KUKA KRL program: EPS_2_251806_MH48A_A_20260212042246.src

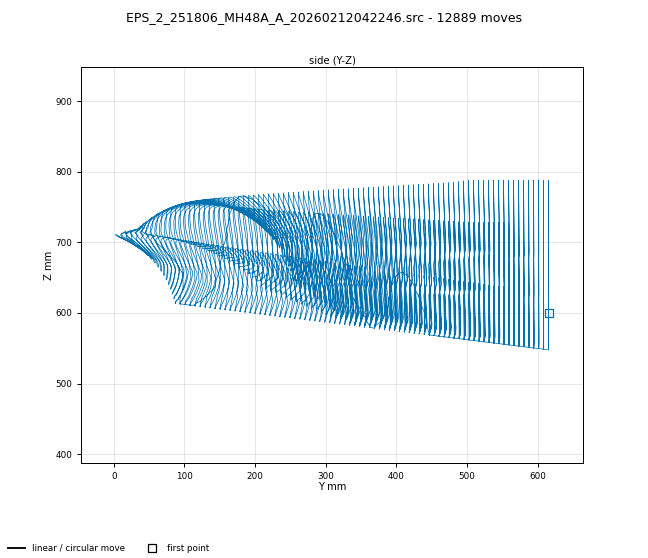
[picture p0: tool path of EPS_2_251806_MH48A_A_20260212042246.src, 12889 of 12891 moves have a stored position in this frame; points joined in program order, loops and branches not executed]
&ACCESS RVP
&REL 4
&COMMENT QRS 19112012
&PARAM EDITMASK = *
DEF PART()
EXT BAS (BAS_COMMAND :IN,REAL :IN )
INT I
BAS (#INITMOV,0 )

;KUKA QRS Post kuka4.cps  Date:22-06-2017 !

File_ID=3020

QRS_PRE_INIT()

;Init var - Until changes are made in qrs_pre_init
Outlet_Square_prg=0
Inlet_1_Square_prg=0
Inlet_2_Square_prg=0
Inlet_3_Square_prg=0
Inlet_4_Square_prg=0
Inlet_5_Square_prg=0

Outlet_1={X 0.000, Y 504.220, Z 687.500, B 0.000, E1 0.000 }
Inlet_1={X 0.000, Y 539.050, Z 207.500, B 0.000, E1 194.000 }
Inlet_2={X 0.000, Y 508.580, Z 627.500, B 0.000, E1 257.000 }
Outlet_1_type=201
Inlet_1_type=201
Inlet_2_type=201
;QRS#1=Sidecore dimensions
;QRS#2=200-8" PVC SDR 35
;QRS#3=200-8" PVC SDR 35
;QRS#4=200-8" PVC SDR 35
;QRS#5=
;QRS#6=
;QRS#7=
;QRS#8=
;QRS#9=12-08 PSX
;QRS#10=12-08 PSX
;QRS#11=12-08 PSX
;QRS#12=
;QRS#13=
;QRS#14=
;QRS#15=
;QRS#16=1220x127x1067 3,5'
;QRS#17=EPS Height
;QRS#18=788
;QRS#19=*
;QRS#20= UPDATED VERSION 22-06-2017
;QRS#21=*
Outlet_Square=0100
Inlet_1_Square=0100
Inlet_2_Square=0100
Inlet_3_Square=0
Inlet_4_Square=0
Inlet_5_Square=0
Mill_Square=1
Outlet_Square_Prg=204
Inlet_1_Square_prg=204
Inlet_2_Square_prg=204

QRS_INIT()

$ADVANCE=5

; T1
PTP {E1 173.607,E2 173.607}
PTP {X 0,Y 615.504,A -85,B 0,C 180,E1 173.607,E2 173.607,E3 0,E4 0,E5 0,E6 0}
QRS_SPEED_INIT()
LIN {X 0,Y 615.504,Z 600,A -85,B 0,C 180,E1 173.607,E2 173.607,E3 0,E4 0,E5 0,E6 0} C_VEL
LIN {X 0,Y 615.504,Z 557.872,A -85,B 0,C 180,E1 173.607,E2 173.607} C_VEL
LIN {X 0,Y 615.504,Z 549.695,A -85,B 0,C 180,E1 173.607,E2 173.607} C_VEL
LIN {X 0,Y 615.491,Z 547.695,A -85,B 0,C 180,E1 173.421,E2 173.421} C_VEL
LIN {X 0,Y 615.488,Z 547.7,A -85,B 0,C 180,E1 170.801,E2 170.801} C_VEL
LIN {X 0,Y 615.487,Z 547.699,A -85,B 0,C 180,E1 168.139,E2 168.139} C_VEL
LIN {X 0,Y 615.487,Z 547.696,A -85,B 0,C 180,E1 165.451,E2 165.451} C_VEL
LIN {X 0,Y 615.478,Z 547.7,A -85,B 0,C 180,E1 162.73,E2 162.73} C_VEL
LIN {X 0,Y 615.483,Z 547.7,A -85,B 0,C 180,E1 159.967,E2 159.967} C_VEL
LIN {X 0,Y 615.482,Z 547.697,A -85,B 0,C 180,E1 157.156,E2 157.156} C_VEL
LIN {X 0,Y 615.498,Z 547.7,A -85,B 0,C 180,E1 154.285,E2 154.285} C_VEL
LIN {X 0,Y 615.485,Z 547.696,A -85,B 0,C 180,E1 151.342,E2 151.342} C_VEL
LIN {X 0,Y 615.477,Z 547.698,A -85,B 0,C 180,E1 148.916,E2 148.916} C_VEL
LIN {X 0,Y 615.486,Z 547.697,A -85,B 0,C 180,E1 146.466,E2 146.466} C_VEL
LIN {X 0,Y 615.491,Z 547.698,A -85,B 0,C 180,E1 143.576,E2 143.576} C_VEL
LIN {X 0,Y 615.479,Z 547.698,A -85,B 0,C 180,E1 140.939,E2 140.939} C_VEL
LIN {X 0,Y 615.486,Z 547.696,A -85,B 0,C 180,E1 138.526,E2 138.526} C_VEL
LIN {X 0,Y 615.489,Z 547.698,A -85,B 0,C 180,E1 135.851,E2 135.851} C_VEL
LIN {X 0,Y 615.486,Z 547.699,A -85,B 0,C 180,E1 133.048,E2 133.048} C_VEL
LIN {X 0,Y 615.496,Z 547.695,A -85,B 0,C 180,E1 130.09,E2 130.09} C_VEL
LIN {X 0,Y 615.495,Z 547.697,A -85,B 0,C 180,E1 127.242,E2 127.242} C_VEL
LIN {X 0,Y 615.479,Z 547.698,A -85,B 0,C 180,E1 124.7,E2 124.7} C_VEL
LIN {X 0,Y 615.494,Z 547.695,A -85,B 0,C 180,E1 122.332,E2 122.332} C_VEL
LIN {X 0,Y 615.486,Z 547.7,A -85,B 0,C 180,E1 119.407,E2 119.407} C_VEL
LIN {X 0,Y 615.491,Z 547.699,A -85,B 0,C 180,E1 117.046,E2 117.046} C_VEL
LIN {X 0,Y 615.495,Z 547.695,A -85,B 0,C 180,E1 114.272,E2 114.272} C_VEL
LIN {X 0,Y 615.48,Z 547.699,A -85,B 0,C 180,E1 111.433,E2 111.433} C_VEL
LIN {X 0,Y 615.489,Z 547.699,A -85,B 0,C 180,E1 108.606,E2 108.606} C_VEL
LIN {X 0,Y 615.489,Z 547.695,A -85,B 0,C 180,E1 105.906,E2 105.906} C_VEL
LIN {X 0,Y 615.488,Z 547.697,A -85,B 0,C 180,E1 103.202,E2 103.202} C_VEL
LIN {X 0,Y 615.491,Z 547.701,A -85,B 0,C 180,E1 100.527,E2 100.527} C_VEL
LIN {X 0,Y 615.487,Z 547.697,A -85,B 0,C 180,E1 97.876,E2 97.876} C_VEL
LIN {X 0,Y 615.481,Z 547.697,A -85,B 0,C 180,E1 95.242,E2 95.242} C_VEL
LIN {X 0,Y 615.483,Z 547.699,A -85,B 0,C 180,E1 92.618,E2 92.618} C_VEL
LIN {X 0,Y 615.487,Z 547.702,A -85,B 0,C 180,E1 90.001,E2 90.001} C_VEL
LIN {X 0,Y 615.482,Z 547.697,A -85,B 0,C 180,E1 87.239,E2 87.239} C_VEL
LIN {X 0,Y 615.486,Z 560.488,A -85,B 0,C 180,E1 86.81,E2 86.81} C_VEL
LIN {X 0,Y 615.491,Z 571.428,A -85,B 0,C 180,E1 86.318,E2 86.318} C_VEL
LIN {X 0,Y 615.49,Z 582.825,A -85,B 0,C 180,E1 85.662,E2 85.662} C_VEL
LIN {X 0,Y 615.498,Z 593.104,A -85,B 0,C 180,E1 84.924,E2 84.924} C_VEL
LIN {X 0,Y 615.5,Z 602.425,A -85,B 0,C 180,E1 84.102,E2 84.102} C_VEL
LIN {X 0,Y 615.496,Z 611.553,A -85,B 0,C 180,E1 83.099,E2 83.099} C_VEL
LIN {X 0,Y 615.497,Z 618.702,A -85,B 0,C 180,E1 82.125,E2 82.125} C_VEL
LIN {X 0,Y 615.496,Z 624.55,A -85,B 0,C 180,E1 81.133,E2 81.133} C_VEL
LIN {X 0,Y 615.497,Z 629.163,A -85,B 0,C 180,E1 80.139,E2 80.139} C_VEL
LIN {X 0,Y 615.495,Z 632.786,A -85,B 0,C 180,E1 79.107,E2 79.107} C_VEL
LIN {X 0,Y 615.496,Z 635.183,A -85,B 0,C 180,E1 78.14,E2 78.14} C_VEL
LIN {X 0,Y 615.495,Z 636.336,A -85,B 0,C 180,E1 77.471,E2 77.471} C_VEL
LIN {X 0,Y 615.495,Z 637.353,A -85,B 0,C 180,E1 76.127,E2 76.127} C_VEL
LIN {X 0,Y 615.497,Z 637.272,A -85,B 0,C 180,E1 75.452,E2 75.452} C_VEL
LIN {X 0,Y 615.496,Z 636.732,A -85,B 0,C 180,E1 74.775,E2 74.775} C_VEL
LIN {X 0,Y 615.493,Z 634.742,A -85,B 0,C 180,E1 73.566,E2 73.566} C_VEL
LIN {X 0,Y 615.496,Z 631.457,A -85,B 0,C 180,E1 72.388,E2 72.388} C_VEL
LIN {X 0,Y 615.497,Z 627.375,A -85,B 0,C 180,E1 71.355,E2 71.355} C_VEL
LIN {X 0,Y 615.497,Z 620.947,A -85,B 0,C 180,E1 70.142,E2 70.142} C_VEL
LIN {X 0,Y 615.497,Z 613.808,A -85,B 0,C 180,E1 69.095,E2 69.095} C_VEL
LIN {X 0,Y 615.499,Z 606.411,A -85,B 0,C 180,E1 68.218,E2 68.218} C_VEL
LIN {X 0,Y 615.5,Z 598.09,A -85,B 0,C 180,E1 67.404,E2 67.404} C_VEL
LIN {X 0,Y 615.5,Z 588.32,A -85,B 0,C 180,E1 66.623,E2 66.623} C_VEL
LIN {X 0,Y 615.496,Z 577.54,A -85,B 0,C 180,E1 65.925,E2 65.925} C_VEL
LIN {X 0,Y 615.491,Z 565.819,A -85,B 0,C 180,E1 65.325,E2 65.325} C_VEL
LIN {X 0,Y 615.487,Z 553.967,A -85,B 0,C 180,E1 64.865,E2 64.865} C_VEL
LIN {X 0,Y 615.479,Z 547.698,A -85,B 0,C 180,E1 64.667,E2 64.667} C_VEL
LIN {X 0,Y 615.484,Z 547.699,A -85,B 0,C 180,E1 62.086,E2 62.086} C_VEL
LIN {X 0,Y 615.499,Z 547.695,A -85,B 0,C 180,E1 59.842,E2 59.842} C_VEL
LIN {X 0,Y 615.491,Z 547.696,A -85,B 0,C 180,E1 57.544,E2 57.544} C_VEL
LIN {X 0,Y 615.478,Z 547.699,A -85,B 0,C 180,E1 55.185,E2 55.185} C_VEL
LIN {X 0,Y 615.494,Z 547.697,A -85,B 0,C 180,E1 52.759,E2 52.759} C_VEL
LIN {X 0,Y 615.494,Z 547.696,A -85,B 0,C 180,E1 49.91,E2 49.91} C_VEL
LIN {X 0,Y 615.482,Z 547.787,A -85,B 0,C 180,E1 48.147,E2 48.147} C_VEL
LIN {X 0,Y 615.494,Z 554.573,A -85,B 0,C 180,E1 45.852,E2 45.852} C_VEL
LIN {X 0,Y 615.482,Z 562.723,A -85,B 0,C 180,E1 43.048,E2 43.048} C_VEL
LIN {X 0,Y 615.484,Z 570.001,A -85,B 0,C 180,E1 40.606,E2 40.606} C_VEL
LIN {X 0,Y 615.48,Z 577.917,A -85,B 0,C 180,E1 38.013,E2 38.013} C_VEL
LIN {X 0,Y 615.478,Z 586.629,A -85,B 0,C 180,E1 35.215,E2 35.215} C_VEL
LIN {X 0,Y 615.484,Z 595.394,A -85,B 0,C 180,E1 32.457,E2 32.457} C_VEL
LIN {X 0,Y 615.498,Z 603.966,A -85,B 0,C 180,E1 29.798,E2 29.798} C_VEL
LIN {X 0,Y 615.478,Z 612.988,A -85,B 0,C 180,E1 27.045,E2 27.045} C_VEL
LIN {X 0,Y 615.492,Z 621.119,A -85,B 0,C 180,E1 24.586,E2 24.586} C_VEL
LIN {X 0,Y 615.492,Z 634.761,A -85,B 0,C 180,E1 24.316,E2 24.316} C_VEL
LIN {X 0,Y 615.486,Z 646.624,A -85,B 0,C 180,E1 23.953,E2 23.953} C_VEL
LIN {X 0,Y 615.484,Z 658.337,A -85,B 0,C 180,E1 23.467,E2 23.467} C_VEL
LIN {X 0,Y 615.481,Z 669.928,A -85,B 0,C 180,E1 22.844,E2 22.844} C_VEL
LIN {X 0,Y 615.499,Z 680.403,A -85,B 0,C 180,E1 22.136,E2 22.136} C_VEL
LIN {X 0,Y 615.497,Z 690.798,A -85,B 0,C 180,E1 21.256,E2 21.256} C_VEL
LIN {X 0,Y 615.496,Z 699.931,A -85,B 0,C 180,E1 20.297,E2 20.297} C_VEL
LIN {X 0,Y 615.498,Z 707.268,A -85,B 0,C 180,E1 19.337,E2 19.337} C_VEL
LIN {X 0,Y 615.498,Z 713.727,A -85,B 0,C 180,E1 18.283,E2 18.283} C_VEL
LIN {X 0,Y 615.495,Z 718.599,A -85,B 0,C 180,E1 17.27,E2 17.27} C_VEL
LIN {X 0,Y 615.495,Z 721.729,A -85,B 0,C 180,E1 16.437,E2 16.437} C_VEL
LIN {X 0,Y 615.496,Z 724.998,A -85,B 0,C 180,E1 15.226,E2 15.226} C_VEL
LIN {X 0,Y 615.494,Z 726.224,A -85,B 0,C 180,E1 14.549,E2 14.549} C_VEL
LIN {X 0,Y 615.494,Z 726.988,A -85,B 0,C 180,E1 13.874,E2 13.874} C_VEL
LIN {X 0,Y 615.494,Z 727.294,A -85,B 0,C 180,E1 12.53,E2 12.53} C_VEL
LIN {X 0,Y 615.495,Z 726.833,A -85,B 0,C 180,E1 11.86,E2 11.86} C_VEL
LIN {X 0,Y 615.493,Z 725.447,A -85,B 0,C 180,E1 10.896,E2 10.896} C_VEL
LIN {X 0,Y 615.499,Z 721.91,A -85,B 0,C 180,E1 9.53,E2 9.53} C_VEL
LIN {X 0,Y 615.495,Z 718.153,A -85,B 0,C 180,E1 8.536,E2 8.536} C_VEL
LIN {X 0,Y 615.498,Z 713.28,A -85,B 0,C 180,E1 7.545,E2 7.545} C_VEL
LIN {X 0,Y 615.496,Z 707.157,A -85,B 0,C 180,E1 6.556,E2 6.556} C_VEL
LIN {X 0,Y 615.499,Z 699.561,A -85,B 0,C 180,E1 5.569,E2 5.569} C_VEL
LIN {X 0,Y 615.497,Z 690.049,A -85,B 0,C 180,E1 4.584,E2 4.584} C_VEL
LIN {X 0,Y 615.5,Z 680.271,A -85,B 0,C 180,E1 3.764,E2 3.764} C_VEL
LIN {X 0,Y 615.479,Z 669.277,A -85,B 0,C 180,E1 3.027,E2 3.027} C_VEL
LIN {X 0,Y 615.489,Z 658.562,A -85,B 0,C 180,E1 2.454,E2 2.454} C_VEL
LIN {X 0,Y 615.477,Z 646.799,A -85,B 0,C 180,E1 1.963,E2 1.963} C_VEL
LIN {X 0,Y 615.487,Z 634.805,A -85,B 0,C 180,E1 1.595,E2 1.595} C_VEL
LIN {X 0,Y 615.488,Z 622.794,A -85,B 0,C 180,E1 1.349,E2 1.349} C_VEL
LIN {X 0,Y 615.485,Z 621.087,A -85,B 0,C 180,E1 1.308,E2 1.308} C_VEL
LIN {X 0,Y 615.485,Z 612.466,A -85,B 0,C 180,E1 -1.309,E2 -1.309} C_VEL
LIN {X 0,Y 615.49,Z 603.925,A -85,B 0,C 180,E1 -3.929,E2 -3.929} C_VEL
LIN {X 0,Y 615.489,Z 595.382,A -85,B 0,C 180,E1 -6.589,E2 -6.589} C_VEL
LIN {X 0,Y 615.496,Z 586.076,A -85,B 0,C 180,E1 -9.53,E2 -9.53} C_VEL
LIN {X 0,Y 615.475,Z 577.824,A -85,B 0,C 180,E1 -12.196,E2 -12.196} C_VEL
LIN {X 0,Y 615.492,Z 569.65,A -85,B 0,C 180,E1 -14.887,E2 -14.887} C_VEL
LIN {X 0,Y 615.499,Z 561.583,A -85,B 0,C 180,E1 -17.613,E2 -17.613} C_VEL
LIN {X 0,Y 615.489,Z 553.106,A -85,B 0,C 180,E1 -20.56,E2 -20.56} C_VEL
LIN {X 0,Y 615.497,Z 549.253,A -85,B 0,C 180,E1 -21.784,E2 -21.784} C_VEL
LIN {X 0,Y 615.484,Z 547.698,A -85,B 0,C 180,E1 -22.243,E2 -22.243} C_VEL
LIN {X 0,Y 615.492,Z 547.701,A -85,B 0,C 180,E1 -24.992,E2 -24.992} C_VEL
LIN {X 0,Y 615.492,Z 547.699,A -85,B 0,C 180,E1 -27.915,E2 -27.915} C_VEL
LIN {X 0,Y 615.5,Z 547.7,A -85,B 0,C 180,E1 -30.16,E2 -30.16} C_VEL
LIN {X 0,Y 615.495,Z 547.697,A -85,B 0,C 180,E1 -32.457,E2 -32.457} C_VEL
LIN {X 0,Y 615.494,Z 547.696,A -85,B 0,C 180,E1 -34.815,E2 -34.815} C_VEL
LIN {X 0,Y 615.49,Z 547.699,A -85,B 0,C 180,E1 -37.242,E2 -37.242} C_VEL
LIN {X 0,Y 615.479,Z 547.699,A -85,B 0,C 180,E1 -40.09,E2 -40.09} C_VEL
LIN {X 0,Y 615.485,Z 547.699,A -85,B 0,C 180,E1 -42.354,E2 -42.354} C_VEL
LIN {X 0,Y 615.481,Z 547.699,A -85,B 0,C 180,E1 -45.069,E2 -45.069} C_VEL
LIN {X 0,Y 615.488,Z 547.7,A -85,B 0,C 180,E1 -47.92,E2 -47.92} C_VEL
LIN {X 0,Y 615.48,Z 547.699,A -85,B 0,C 180,E1 -50.25,E2 -50.25} C_VEL
LIN {X 0,Y 615.49,Z 547.7,A -85,B 0,C 180,E1 -53.063,E2 -53.063} C_VEL
LIN {X 0,Y 615.484,Z 547.718,A -85,B 0,C 180,E1 -54.486,E2 -54.486} C_VEL
LIN {X 0,Y 615.49,Z 561.14,A -85,B 0,C 180,E1 -57.155,E2 -57.155} C_VEL
LIN {X 0,Y 615.499,Z 574.889,A -85,B 0,C 180,E1 -59.842,E2 -59.842} C_VEL
LIN {X 0,Y 615.488,Z 590.604,A -85,B 0,C 180,E1 -62.824,E2 -62.824} C_VEL
LIN {X 0,Y 615.488,Z 606.309,A -85,B 0,C 180,E1 -65.729,E2 -65.729} C_VEL
LIN {X 0,Y 615.486,Z 622.001,A -85,B 0,C 180,E1 -68.569,E2 -68.569} C_VEL
LIN {X 0,Y 615.479,Z 637.926,A -85,B 0,C 180,E1 -71.399,E2 -71.399} C_VEL
LIN {X 0,Y 615.495,Z 653.333,A -85,B 0,C 180,E1 -74.096,E2 -74.096} C_VEL
LIN {X 0,Y 615.488,Z 668.981,A -85,B 0,C 180,E1 -76.8,E2 -76.8} C_VEL
LIN {X 0,Y 615.478,Z 678,A -85,B 0,C 180,E1 -78.328,E2 -78.328} C_VEL
LIN {X 0,Y 615.478,Z 691.273,A -85,B 0,C 180,E1 -78.557,E2 -78.557} C_VEL
LIN {X 0,Y 615.499,Z 704.348,A -85,B 0,C 180,E1 -78.923,E2 -78.923} C_VEL
LIN {X 0,Y 615.476,Z 716.143,A -85,B 0,C 180,E1 -79.384,E2 -79.384} C_VEL
LIN {X 0,Y 615.488,Z 727.587,A -85,B 0,C 180,E1 -79.972,E2 -79.972} C_VEL
LIN {X 0,Y 615.499,Z 739.031,A -85,B 0,C 180,E1 -80.719,E2 -80.719} C_VEL
LIN {X 0,Y 615.498,Z 748.265,A -85,B 0,C 180,E1 -81.464,E2 -81.464} C_VEL
LIN {X 0,Y 615.499,Z 756.659,A -85,B 0,C 180,E1 -82.29,E2 -82.29} C_VEL
LIN {X 0,Y 615.497,Z 764.692,A -85,B 0,C 180,E1 -83.259,E2 -83.259} C_VEL
LIN {X 0,Y 615.498,Z 770.427,A -85,B 0,C 180,E1 -84.102,E2 -84.102} C_VEL
LIN {X 0,Y 615.497,Z 775.875,A -85,B 0,C 180,E1 -85.088,E2 -85.088} C_VEL
LIN {X 0,Y 615.496,Z 780.143,A -85,B 0,C 180,E1 -86.072,E2 -86.072} C_VEL
LIN {X 0,Y 615.495,Z 782.401,A -85,B 0,C 180,E1 -86.728,E2 -86.728} C_VEL
LIN {X 0,Y 615.497,Z 784.234,A -85,B 0,C 180,E1 -87.383,E2 -87.383} C_VEL
LIN {X 0,Y 615.496,Z 785.609,A -85,B 0,C 180,E1 -88.038,E2 -88.038} C_VEL
LIN {X 0,Y 615.496,Z 787.174,A -85,B 0,C 180,E1 -89.346,E2 -89.346} C_VEL
LIN {X 0,Y 615.494,Z 787.389,A -85,B 0,C 180,E1 -90.001,E2 -90.001} C_VEL
LIN {X 0,Y 615.496,Z 786.579,A -85,B 0,C 180,E1 -91.309,E2 -91.309} C_VEL
LIN {X 0,Y 615.496,Z 785.607,A -85,B 0,C 180,E1 -91.964,E2 -91.964} C_VEL
LIN {X 0,Y 615.497,Z 784.231,A -85,B 0,C 180,E1 -92.618,E2 -92.618} C_VEL
LIN {X 0,Y 615.496,Z 781.348,A -85,B 0,C 180,E1 -93.601,E2 -93.601} C_VEL
LIN {X 0,Y 615.498,Z 777.439,A -85,B 0,C 180,E1 -94.585,E2 -94.585} C_VEL
LIN {X 0,Y 615.499,Z 772.402,A -85,B 0,C 180,E1 -95.57,E2 -95.57} C_VEL
LIN {X 0,Y 615.497,Z 765.87,A -85,B 0,C 180,E1 -96.583,E2 -96.583} C_VEL
LIN {X 0,Y 615.497,Z 758.128,A -85,B 0,C 180,E1 -97.546,E2 -97.546} C_VEL
LIN {X 0,Y 615.498,Z 750.039,A -85,B 0,C 180,E1 -98.372,E2 -98.372} C_VEL
LIN {X 0,Y 615.499,Z 740.16,A -85,B 0,C 180,E1 -99.199,E2 -99.199} C_VEL
LIN {X 0,Y 615.486,Z 728.973,A -85,B 0,C 180,E1 -99.946,E2 -99.946} C_VEL
LIN {X 0,Y 615.476,Z 718.013,A -85,B 0,C 180,E1 -100.528,E2 -100.528} C_VEL
LIN {X 0,Y 615.497,Z 705.495,A -85,B 0,C 180,E1 -101.04,E2 -101.04} C_VEL
LIN {X 0,Y 615.479,Z 693.044,A -85,B 0,C 180,E1 -101.402,E2 -101.402} C_VEL
LIN {X 0,Y 615.477,Z 679.431,A -85,B 0,C 180,E1 -101.653,E2 -101.653} C_VEL
LIN {X 0,Y 615.478,Z 677.795,A -85,B 0,C 180,E1 -101.694,E2 -101.694} C_VEL
LIN {X 0,Y 615.491,Z 663.028,A -85,B 0,C 180,E1 -104.24,E2 -104.24} C_VEL
LIN {X 0,Y 615.487,Z 647.605,A -85,B 0,C 180,E1 -106.929,E2 -106.929} C_VEL
LIN {X 0,Y 615.476,Z 632.002,A -85,B 0,C 180,E1 -109.686,E2 -109.686} C_VEL
LIN {X 0,Y 615.48,Z 617.194,A -85,B 0,C 180,E1 -112.344,E2 -112.344} C_VEL
LIN {X 0,Y 615.494,Z 602.704,A -85,B 0,C 180,E1 -114.992,E2 -114.992} C_VEL
LIN {X 0,Y 615.48,Z 589.015,A -85,B 0,C 180,E1 -117.546,E2 -117.546} C_VEL
LIN {X 0,Y 615.499,Z 575.32,A -85,B 0,C 180,E1 -120.16,E2 -120.16} C_VEL
LIN {X 0,Y 615.491,Z 561.625,A -85,B 0,C 180,E1 -122.846,E2 -122.846} C_VEL
LIN {X 0,Y 615.475,Z 547.698,A -85,B 0,C 180,E1 -125.644,E2 -125.644} C_VEL
LIN {X 0,Y 615.489,Z 547.695,A -85,B 0,C 180,E1 -128.069,E2 -128.069} C_VEL
LIN {X 0,Y 615.481,Z 547.698,A -85,B 0,C 180,E1 -130.607,E2 -130.607} C_VEL
LIN {X 0,Y 615.499,Z 547.7,A -85,B 0,C 180,E1 -133.244,E2 -133.244} C_VEL
LIN {X 0,Y 615.485,Z 547.697,A -85,B 0,C 180,E1 -136.003,E2 -136.003} C_VEL
LIN {X 0,Y 615.486,Z 547.699,A -85,B 0,C 180,E1 -138.906,E2 -138.906} C_VEL
LIN {X 0,Y 615.484,Z 547.698,A -85,B 0,C 180,E1 -141.095,E2 -141.095} C_VEL
LIN {X 0,Y 615.495,Z 547.697,A -85,B 0,C 180,E1 -143.575,E2 -143.575} C_VEL
LIN {X 0,Y 615.489,Z 547.699,A -85,B 0,C 180,E1 -145.978,E2 -145.978} C_VEL
LIN {X 0,Y 615.49,Z 547.699,A -85,B 0,C 180,E1 -148.314,E2 -148.314} C_VEL
LIN {X 0,Y 615.482,Z 547.7,A -85,B 0,C 180,E1 -150.593,E2 -150.593} C_VEL
LIN {X 0,Y 615.487,Z 547.699,A -85,B 0,C 180,E1 -152.955,E2 -152.955} C_VEL
LIN {X 0,Y 615.482,Z 547.699,A -85,B 0,C 180,E1 -155.727,E2 -155.727} C_VEL
LIN {X 0,Y 615.486,Z 547.697,A -85,B 0,C 180,E1 -158.568,E2 -158.568} C_VEL
LIN {X 0,Y 615.493,Z 547.7,A -85,B 0,C 180,E1 -161.394,E2 -161.394} C_VEL
LIN {X 0,Y 615.48,Z 547.698,A -85,B 0,C 180,E1 -164.094,E2 -164.094} C_VEL
LIN {X 0,Y 615.479,Z 547.699,A -85,B 0,C 180,E1 -166.798,E2 -166.798} C_VEL
LIN {X 0,Y 615.49,Z 547.702,A -85,B 0,C 180,E1 -169.473,E2 -169.473} C_VEL
LIN {X 0,Y 615.483,Z 547.698,A -85,B 0,C 180,E1 -172.124,E2 -172.124} C_VEL
LIN {X 0,Y 615.481,Z 547.697,A -85,B 0,C 180,E1 -174.758,E2 -174.758} C_VEL
LIN {X 0,Y 615.492,Z 547.697,A -85,B 0,C 180,E1 -177.382,E2 -177.382} C_VEL
LIN {X 0,Y 615.489,Z 547.703,A -85,B 0,C 180,E1 -180,E2 -180} C_VEL
LIN {X 0,Y 615.492,Z 547.697,A -85,B 0,C 180,E1 -182.618,E2 -182.618} C_VEL
LIN {X 0,Y 615.481,Z 547.697,A -85,B 0,C 180,E1 -185.241,E2 -185.241} C_VEL
LIN {X 0,Y 615.491,Z 547.695,A -85,B 0,C 180,E1 -186.579,E2 -186.579} C_VEL
LIN {X 0,Y 614.815,Z 547.844,A -85,B 0,C 180,E1 -187.125,E2 -187.125} C_VEL
LIN {X 0,Y 611.981,Z 548.257,A -85,B 0,C 180,E1 -188.011,E2 -188.011} C_VEL
LIN {X 0,Y 609.587,Z 548.568,A -85,B 0,C 180,E1 -188.724,E2 -188.724} C_VEL
LIN {X 0,Y 608.549,Z 548.687,A -85,B 0,C 180,E1 -189.273,E2 -189.273} C_VEL
LIN {X 0,Y 608.458,Z 548.696,A -85,B 0,C 180,E1 -189.46,E2 -189.46} C_VEL
LIN {X 0,Y 608.464,Z 548.694,A -85,B 0,C 180,E1 -191.999,E2 -191.999} C_VEL
LIN {X 0,Y 608.478,Z 548.692,A -85,B 0,C 180,E1 -194.72,E2 -194.72} C_VEL
LIN {X 0,Y 608.446,Z 548.699,A -85,B 0,C 180,E1 -197.476,E2 -197.476} C_VEL
LIN {X 0,Y 608.45,Z 548.696,A -85,B 0,C 180,E1 -199.57,E2 -199.57} C_VEL
LIN {X 0,Y 608.46,Z 548.695,A -85,B 0,C 180,E1 -202.476,E2 -202.476} C_VEL
LIN {X 0,Y 608.45,Z 548.698,A -85,B 0,C 180,E1 -204.571,E2 -204.571} C_VEL
LIN {X 0,Y 608.481,Z 548.692,A -85,B 0,C 180,E1 -207.207,E2 -207.207} C_VEL
LIN {X 0,Y 608.471,Z 548.693,A -85,B 0,C 180,E1 -209.972,E2 -209.972} C_VEL
LIN {X 0,Y 608.453,Z 548.696,A -85,B 0,C 180,E1 -212.879,E2 -212.879} C_VEL
LIN {X 0,Y 608.449,Z 548.696,A -85,B 0,C 180,E1 -215.277,E2 -215.277} C_VEL
LIN {X 0,Y 608.469,Z 548.693,A -85,B 0,C 180,E1 -217.746,E2 -217.746} C_VEL
LIN {X 0,Y 608.446,Z 548.695,A -85,B 0,C 180,E1 -220.328,E2 -220.328} C_VEL
LIN {X 0,Y 608.453,Z 548.696,A -85,B 0,C 180,E1 -222.959,E2 -222.959} C_VEL
LIN {X 0,Y 608.46,Z 548.695,A -85,B 0,C 180,E1 -225.735,E2 -225.735} C_VEL
LIN {X 0,Y 608.464,Z 548.694,A -85,B 0,C 180,E1 -228.657,E2 -228.657} C_VEL
LIN {X 0,Y 608.469,Z 548.696,A -85,B 0,C 180,E1 -231.412,E2 -231.412} C_VEL
LIN {X 0,Y 608.445,Z 548.697,A -85,B 0,C 180,E1 -233.954,E2 -233.954} C_VEL
LIN {X 0,Y 608.463,Z 548.694,A -85,B 0,C 180,E1 -236.329,E2 -236.329} C_VEL
LIN {X 0,Y 608.479,Z 548.692,A -85,B 0,C 180,E1 -238.727,E2 -238.727} C_VEL
LIN {X 0,Y 608.467,Z 548.693,A -85,B 0,C 180,E1 -241.381,E2 -241.381} C_VEL
LIN {X 0,Y 608.451,Z 548.696,A -85,B 0,C 180,E1 -243.964,E2 -243.964} C_VEL
LIN {X 0,Y 608.472,Z 548.692,A -85,B 0,C 180,E1 -246.155,E2 -246.155} C_VEL
LIN {X 0,Y 608.468,Z 548.693,A -85,B 0,C 180,E1 -248.308,E2 -248.308} C_VEL
LIN {X 0,Y 608.473,Z 548.696,A -85,B 0,C 180,E1 -251.283,E2 -251.283} C_VEL
LIN {X 0,Y 608.464,Z 548.694,A -85,B 0,C 180,E1 -253.906,E2 -253.906} C_VEL
LIN {X 0,Y 608.465,Z 548.693,A -85,B 0,C 180,E1 -256.643,E2 -256.643} C_VEL
LIN {X 0,Y 608.468,Z 548.695,A -85,B 0,C 180,E1 -259.35,E2 -259.35} C_VEL
LIN {X 0,Y 608.478,Z 548.693,A -85,B 0,C 180,E1 -262.033,E2 -262.033} C_VEL
LIN {X 0,Y 608.462,Z 548.693,A -85,B 0,C 180,E1 -264.698,E2 -264.698} C_VEL
LIN {X 0,Y 608.475,Z 548.693,A -85,B 0,C 180,E1 -267.351,E2 -267.351} C_VEL
LIN {X 0,Y 608.478,Z 548.695,A -85,B 0,C 180,E1 -269.999,E2 -269.999} C_VEL
LIN {X 0,Y 608.472,Z 548.693,A -85,B 0,C 180,E1 -272.647,E2 -272.647} C_VEL
LIN {X 0,Y 608.506,Z 562.528,A -85,B 0,C 180,E1 -273.144,E2 -273.144} C_VEL
LIN {X 0,Y 608.512,Z 574.619,A -85,B 0,C 180,E1 -273.724,E2 -273.724} C_VEL
LIN {X 0,Y 608.479,Z 585.509,A -85,B 0,C 180,E1 -274.388,E2 -274.388} C_VEL
LIN {X 0,Y 608.482,Z 595.356,A -85,B 0,C 180,E1 -275.135,E2 -275.135} C_VEL
LIN {X 0,Y 608.456,Z 604.326,A -85,B 0,C 180,E1 -275.966,E2 -275.966} C_VEL
LIN {X 0,Y 608.462,Z 613.118,A -85,B 0,C 180,E1 -276.965,E2 -276.965} C_VEL
LIN {X 0,Y 608.44,Z 620.192,A -85,B 0,C 180,E1 -277.967,E2 -277.967} C_VEL
LIN {X 0,Y 608.446,Z 625.856,A -85,B 0,C 180,E1 -278.97,E2 -278.97} C_VEL
LIN {X 0,Y 608.436,Z 630.327,A -85,B 0,C 180,E1 -279.977,E2 -279.977} C_VEL
LIN {X 0,Y 608.452,Z 633.614,A -85,B 0,C 180,E1 -280.949,E2 -280.949} C_VEL
LIN {X 0,Y 608.439,Z 636.102,A -85,B 0,C 180,E1 -281.999,E2 -281.999} C_VEL
LIN {X 0,Y 608.439,Z 637.765,A -85,B 0,C 180,E1 -283.356,E2 -283.356} C_VEL
LIN {X 0,Y 608.421,Z 638,A -85,B 0,C 180,E1 -284.038,E2 -284.038} C_VEL
LIN {X 0,Y 608.418,Z 637.773,A -85,B 0,C 180,E1 -284.721,E2 -284.721} C_VEL
LIN {X 0,Y 608.419,Z 637.139,A -85,B 0,C 180,E1 -285.407,E2 -285.407} C_VEL
LIN {X 0,Y 608.422,Z 635.208,A -85,B 0,C 180,E1 -286.515,E2 -286.515} C_VEL
LIN {X 0,Y 608.424,Z 632.57,A -85,B 0,C 180,E1 -287.477,E2 -287.477} C_VEL
LIN {X 0,Y 608.431,Z 627.848,A -85,B 0,C 180,E1 -288.706,E2 -288.706} C_VEL
LIN {X 0,Y 608.451,Z 622.485,A -85,B 0,C 180,E1 -289.745,E2 -289.745} C_VEL
LIN {X 0,Y 608.466,Z 615.66,A -85,B 0,C 180,E1 -290.787,E2 -290.787} C_VEL
LIN {X 0,Y 608.455,Z 606.774,A -85,B 0,C 180,E1 -291.869,E2 -291.869} C_VEL
LIN {X 0,Y 608.47,Z 596.855,A -85,B 0,C 180,E1 -292.826,E2 -292.826} C_VEL
LIN {X 0,Y 608.493,Z 586.091,A -85,B 0,C 180,E1 -293.662,E2 -293.662} C_VEL
LIN {X 0,Y 608.495,Z 574.644,A -85,B 0,C 180,E1 -294.365,E2 -294.365} C_VEL
LIN {X 0,Y 608.515,Z 562.849,A -85,B 0,C 180,E1 -294.932,E2 -294.932} C_VEL
LIN {X 0,Y 608.512,Z 550.797,A -85,B 0,C 180,E1 -295.37,E2 -295.37} C_VEL
LIN {X 0,Y 608.454,Z 548.695,A -85,B 0,C 180,E1 -295.446,E2 -295.446} C_VEL
LIN {X 0,Y 608.449,Z 548.695,A -85,B 0,C 180,E1 -297.517,E2 -297.517} C_VEL
LIN {X 0,Y 608.469,Z 548.693,A -85,B 0,C 180,E1 -299.972,E2 -299.972} C_VEL
LIN {X 0,Y 608.464,Z 548.694,A -85,B 0,C 180,E1 -302.523,E2 -302.523} C_VEL
LIN {X 0,Y 608.433,Z 548.699,A -85,B 0,C 180,E1 -305.277,E2 -305.277} C_VEL
LIN {X 0,Y 608.474,Z 548.693,A -85,B 0,C 180,E1 -307.745,E2 -307.745} C_VEL
LIN {X 0,Y 608.475,Z 548.692,A -85,B 0,C 180,E1 -310.332,E2 -310.332} C_VEL
LIN {X 0,Y 608.453,Z 548.695,A -85,B 0,C 180,E1 -311.769,E2 -311.769} C_VEL
LIN {X 0,Y 608.502,Z 556.172,A -85,B 0,C 180,E1 -314.269,E2 -314.269} C_VEL
LIN {X 0,Y 608.503,Z 564.176,A -85,B 0,C 180,E1 -317.045,E2 -317.045} C_VEL
LIN {X 0,Y 608.458,Z 572.042,A -85,B 0,C 180,E1 -319.697,E2 -319.697} C_VEL
LIN {X 0,Y 608.481,Z 579.797,A -85,B 0,C 180,E1 -322.255,E2 -322.255} C_VEL
LIN {X 0,Y 608.452,Z 588.597,A -85,B 0,C 180,E1 -325.092,E2 -325.092} C_VEL
LIN {X 0,Y 608.436,Z 597.489,A -85,B 0,C 180,E1 -327.904,E2 -327.904} C_VEL
LIN {X 0,Y 608.447,Z 606.157,A -85,B 0,C 180,E1 -330.6,E2 -330.6} C_VEL
LIN {X 0,Y 608.418,Z 614.714,A -85,B 0,C 180,E1 -333.225,E2 -333.225} C_VEL
LIN {X 0,Y 608.448,Z 621.484,A -85,B 0,C 180,E1 -335.281,E2 -335.281} C_VEL
LIN {X 0,Y 608.534,Z 635.05,A -85,B 0,C 180,E1 -335.557,E2 -335.557} C_VEL
LIN {X 0,Y 608.51,Z 646.973,A -85,B 0,C 180,E1 -335.927,E2 -335.927} C_VEL
LIN {X 0,Y 608.503,Z 658.842,A -85,B 0,C 180,E1 -336.428,E2 -336.428} C_VEL
LIN {X 0,Y 608.497,Z 670.707,A -85,B 0,C 180,E1 -337.076,E2 -337.076} C_VEL
LIN {X 0,Y 608.491,Z 680.853,A -85,B 0,C 180,E1 -337.774,E2 -337.774} C_VEL
LIN {X 0,Y 608.461,Z 691.268,A -85,B 0,C 180,E1 -338.664,E2 -338.664} C_VEL
LIN {X 0,Y 608.458,Z 700.073,A -85,B 0,C 180,E1 -339.592,E2 -339.592} C_VEL
LIN {X 0,Y 608.45,Z 707.795,A -85,B 0,C 180,E1 -340.605,E2 -340.605} C_VEL
LIN {X 0,Y 608.444,Z 713.664,A -85,B 0,C 180,E1 -341.557,E2 -341.557} C_VEL
LIN {X 0,Y 608.429,Z 718.444,A -85,B 0,C 180,E1 -342.523,E2 -342.523} C_VEL
LIN {X 0,Y 608.426,Z 722.146,A -85,B 0,C 180,E1 -343.481,E2 -343.481} C_VEL
LIN {X 0,Y 608.42,Z 725.248,A -85,B 0,C 180,E1 -344.593,E2 -344.593} C_VEL
LIN {X 0,Y 608.417,Z 726.566,A -85,B 0,C 180,E1 -345.278,E2 -345.278} C_VEL
LIN {X 0,Y 608.432,Z 727.499,A -85,B 0,C 180,E1 -345.993,E2 -345.993} C_VEL
LIN {X 0,Y 608.437,Z 727.912,A -85,B 0,C 180,E1 -346.643,E2 -346.643} C_VEL
LIN {X 0,Y 608.438,Z 727.577,A -85,B 0,C 180,E1 -348,E2 -348} C_VEL
LIN {X 0,Y 608.449,Z 726.172,A -85,B 0,C 180,E1 -349.049,E2 -349.049} C_VEL
LIN {X 0,Y 608.43,Z 722.947,A -85,B 0,C 180,E1 -350.358,E2 -350.358} C_VEL
LIN {X 0,Y 608.427,Z 719.314,A -85,B 0,C 180,E1 -351.364,E2 -351.364} C_VEL
LIN {X 0,Y 608.448,Z 714.57,A -85,B 0,C 180,E1 -352.367,E2 -352.367} C_VEL
LIN {X 0,Y 608.46,Z 707.748,A -85,B 0,C 180,E1 -353.492,E2 -353.492} C_VEL
LIN {X 0,Y 608.461,Z 699.778,A -85,B 0,C 180,E1 -354.532,E2 -354.532} C_VEL
LIN {X 0,Y 608.489,Z 690.17,A -85,B 0,C 180,E1 -355.529,E2 -355.529} C_VEL
LIN {X 0,Y 608.48,Z 680.3,A -85,B 0,C 180,E1 -356.358,E2 -356.358} C_VEL
LIN {X 0,Y 608.489,Z 669.201,A -85,B 0,C 180,E1 -357.104,E2 -357.104} C_VEL
LIN {X 0,Y 608.498,Z 656.676,A -85,B 0,C 180,E1 -357.766,E2 -357.766} C_VEL
LIN {X 0,Y 608.523,Z 644.093,A -85,B 0,C 180,E1 -358.263,E2 -358.263} C_VEL
LIN {X 0,Y 608.542,Z 630.713,A -85,B 0,C 180,E1 -358.635,E2 -358.635} C_VEL
LIN {X 0,Y 608.435,Z 621.464,A -85,B 0,C 180,E1 -358.821,E2 -358.821} C_VEL
LIN {X 0,Y 608.437,Z 613.263,A -85,B 0,C 180,E1 -361.324,E2 -361.324} C_VEL
LIN {X 0,Y 608.442,Z 604.677,A -85,B 0,C 180,E1 -363.974,E2 -363.974} C_VEL
LIN {X 0,Y 608.469,Z 596.182,A -85,B 0,C 180,E1 -366.633,E2 -366.633} C_VEL
LIN {X 0,Y 608.473,Z 587.784,A -85,B 0,C 180,E1 -369.306,E2 -369.306} C_VEL
LIN {X 0,Y 608.457,Z 579.483,A -85,B 0,C 180,E1 -372,E2 -372} C_VEL
LIN {X 0,Y 608.483,Z 571.277,A -85,B 0,C 180,E1 -374.721,E2 -374.721} C_VEL
LIN {X 0,Y 608.502,Z 563.174,A -85,B 0,C 180,E1 -377.475,E2 -377.475} C_VEL
LIN {X 0,Y 608.482,Z 555.18,A -85,B 0,C 180,E1 -380.274,E2 -380.274} C_VEL
LIN {X 0,Y 608.45,Z 548.696,A -85,B 0,C 180,E1 -382.228,E2 -382.228} C_VEL
LIN {X 0,Y 608.455,Z 548.695,A -85,B 0,C 180,E1 -384.571,E2 -384.571} C_VEL
LIN {X 0,Y 608.483,Z 548.693,A -85,B 0,C 180,E1 -387.21,E2 -387.21} C_VEL
LIN {X 0,Y 608.472,Z 548.694,A -85,B 0,C 180,E1 -389.974,E2 -389.974} C_VEL
LIN {X 0,Y 608.468,Z 548.694,A -85,B 0,C 180,E1 -392.525,E2 -392.525} C_VEL
LIN {X 0,Y 608.451,Z 548.698,A -85,B 0,C 180,E1 -395.277,E2 -395.277} C_VEL
LIN {X 0,Y 608.468,Z 548.694,A -85,B 0,C 180,E1 -397.747,E2 -397.747} C_VEL
LIN {X 0,Y 608.452,Z 548.697,A -85,B 0,C 180,E1 -400.33,E2 -400.33} C_VEL
LIN {X 0,Y 608.47,Z 548.694,A -85,B 0,C 180,E1 -403.31,E2 -403.31} C_VEL
LIN {X 0,Y 608.469,Z 548.693,A -85,B 0,C 180,E1 -406.132,E2 -406.132} C_VEL
LIN {X 0,Y 608.453,Z 548.698,A -85,B 0,C 180,E1 -408.824,E2 -408.824} C_VEL
LIN {X 0,Y 608.469,Z 548.693,A -85,B 0,C 180,E1 -411.413,E2 -411.413} C_VEL
LIN {X 0,Y 608.479,Z 548.694,A -85,B 0,C 180,E1 -414.228,E2 -414.228} C_VEL
LIN {X 0,Y 608.477,Z 548.736,A -85,B 0,C 180,E1 -414.319,E2 -414.319} C_VEL
LIN {X 0,Y 608.642,Z 559.175,A -85,B 0,C 180,E1 -416.342,E2 -416.342} C_VEL
LIN {X 0,Y 608.616,Z 571.03,A -85,B 0,C 180,E1 -418.707,E2 -418.707} C_VEL
LIN {X 0,Y 608.585,Z 584.693,A -85,B 0,C 180,E1 -421.361,E2 -421.361} C_VEL
LIN {X 0,Y 608.566,Z 598.461,A -85,B 0,C 180,E1 -423.971,E2 -423.971} C_VEL
LIN {X 0,Y 608.542,Z 614.175,A -85,B 0,C 180,E1 -426.881,E2 -426.881} C_VEL
LIN {X 0,Y 608.502,Z 629.889,A -85,B 0,C 180,E1 -429.728,E2 -429.728} C_VEL
LIN {X 0,Y 608.496,Z 645.603,A -85,B 0,C 180,E1 -432.526,E2 -432.526} C_VEL
LIN {X 0,Y 608.477,Z 661.317,A -85,B 0,C 180,E1 -435.28,E2 -435.28} C_VEL
LIN {X 0,Y 608.451,Z 678.013,A -85,B 0,C 180,E1 -438.17,E2 -438.17} C_VEL
LIN {X 0,Y 608.535,Z 694.125,A -85,B 0,C 180,E1 -438.488,E2 -438.488} C_VEL
LIN {X 0,Y 608.525,Z 707.321,A -85,B 0,C 180,E1 -438.896,E2 -438.896} C_VEL
LIN {X 0,Y 608.504,Z 719.936,A -85,B 0,C 180,E1 -439.436,E2 -439.436} C_VEL
LIN {X 0,Y 608.48,Z 730.59,A -85,B 0,C 180,E1 -440.024,E2 -440.024} C_VEL
LIN {X 0,Y 608.483,Z 741.483,A -85,B 0,C 180,E1 -440.779,E2 -440.779} C_VEL
LIN {X 0,Y 608.475,Z 752.119,A -85,B 0,C 180,E1 -441.699,E2 -441.699} C_VEL
LIN {X 0,Y 608.47,Z 759.966,A -85,B 0,C 180,E1 -442.535,E2 -442.535} C_VEL
LIN {X 0,Y 608.46,Z 767.289,A -85,B 0,C 180,E1 -443.485,E2 -443.485} C_VEL
LIN {X 0,Y 608.45,Z 772.869,A -85,B 0,C 180,E1 -444.366,E2 -444.366} C_VEL
LIN {X 0,Y 608.432,Z 777.953,A -85,B 0,C 180,E1 -445.363,E2 -445.363} C_VEL
LIN {X 0,Y 608.449,Z 781.898,A -85,B 0,C 180,E1 -446.358,E2 -446.358} C_VEL
LIN {X 0,Y 608.425,Z 784.811,A -85,B 0,C 180,E1 -447.352,E2 -447.352} C_VEL
LIN {X 0,Y 608.441,Z 786.202,A -85,B 0,C 180,E1 -448.015,E2 -448.015} C_VEL
LIN {X 0,Y 608.438,Z 787.784,A -85,B 0,C 180,E1 -449.339,E2 -449.339} C_VEL
LIN {X 0,Y 608.434,Z 788,A -85,B 0,C 180,E1 -450.001,E2 -450.001} C_VEL
LIN {X 0,Y 608.448,Z 787.183,A -85,B 0,C 180,E1 -451.324,E2 -451.324} C_VEL
LIN {X 0,Y 608.441,Z 786.2,A -85,B 0,C 180,E1 -451.986,E2 -451.986} C_VEL
LIN {X 0,Y 608.425,Z 784.808,A -85,B 0,C 180,E1 -452.649,E2 -452.649} C_VEL
LIN {X 0,Y 608.449,Z 781.894,A -85,B 0,C 180,E1 -453.643,E2 -453.643} C_VEL
LIN {X 0,Y 608.432,Z 777.948,A -85,B 0,C 180,E1 -454.638,E2 -454.638} C_VEL
LIN {X 0,Y 608.437,Z 771.873,A -85,B 0,C 180,E1 -455.801,E2 -455.801} C_VEL
LIN {X 0,Y 608.462,Z 765.231,A -85,B 0,C 180,E1 -456.8,E2 -456.8} C_VEL
LIN {X 0,Y 608.456,Z 756.984,A -85,B 0,C 180,E1 -457.801,E2 -457.801} C_VEL
LIN {X 0,Y 608.472,Z 748.53,A -85,B 0,C 180,E1 -458.636,E2 -458.636} C_VEL
LIN {X 0,Y 608.48,Z 738.083,A -85,B 0,C 180,E1 -459.474,E2 -459.474} C_VEL
LIN {X 0,Y 608.5,Z 727.746,A -85,B 0,C 180,E1 -460.145,E2 -460.145} C_VEL
LIN {X 0,Y 608.504,Z 716.264,A -85,B 0,C 180,E1 -460.74,E2 -460.74} C_VEL
LIN {X 0,Y 608.533,Z 703.914,A -85,B 0,C 180,E1 -461.224,E2 -461.224} C_VEL
LIN {X 0,Y 608.535,Z 690.416,A -85,B 0,C 180,E1 -461.597,E2 -461.597} C_VEL
LIN {X 0,Y 608.444,Z 678.153,A -85,B 0,C 180,E1 -461.81,E2 -461.81} C_VEL
LIN {X 0,Y 608.464,Z 663.358,A -85,B 0,C 180,E1 -464.379,E2 -464.379} C_VEL
LIN {X 0,Y 608.482,Z 647.707,A -85,B 0,C 180,E1 -467.13,E2 -467.13} C_VEL
LIN {X 0,Y 608.488,Z 632.056,A -85,B 0,C 180,E1 -469.921,E2 -469.921} C_VEL
LIN {X 0,Y 608.532,Z 617.876,A -85,B 0,C 180,E1 -472.492,E2 -472.492} C_VEL
LIN {X 0,Y 608.559,Z 602.71,A -85,B 0,C 180,E1 -475.297,E2 -475.297} C_VEL
LIN {X 0,Y 608.608,Z 587.058,A -85,B 0,C 180,E1 -478.259,E2 -478.259} C_VEL
LIN {X 0,Y 608.602,Z 573.403,A -85,B 0,C 180,E1 -480.915,E2 -480.915} C_VEL
LIN {X 0,Y 608.649,Z 561.625,A -85,B 0,C 180,E1 -483.263,E2 -483.263} C_VEL
LIN {X 0,Y 608.605,Z 551.401,A -85,B 0,C 180,E1 -485.267,E2 -485.267} C_VEL
LIN {X 0,Y 608.459,Z 548.695,A -85,B 0,C 180,E1 -485.836,E2 -485.836} C_VEL
LIN {X 0,Y 608.474,Z 548.696,A -85,B 0,C 180,E1 -488.588,E2 -488.588} C_VEL
LIN {X 0,Y 608.464,Z 548.693,A -85,B 0,C 180,E1 -491.342,E2 -491.342} C_VEL
LIN {X 0,Y 608.461,Z 548.695,A -85,B 0,C 180,E1 -494.264,E2 -494.264} C_VEL
LIN {X 0,Y 608.459,Z 548.695,A -85,B 0,C 180,E1 -497.04,E2 -497.04} C_VEL
LIN {X 0,Y 608.457,Z 548.694,A -85,B 0,C 180,E1 -499.697,E2 -499.697} C_VEL
LIN {X 0,Y 608.482,Z 548.692,A -85,B 0,C 180,E1 -502.841,E2 -502.841} C_VEL
LIN {X 0,Y 608.476,Z 548.692,A -85,B 0,C 180,E1 -505.531,E2 -505.531} C_VEL
LIN {X 0,Y 608.464,Z 548.693,A -85,B 0,C 180,E1 -507.905,E2 -507.905} C_VEL
LIN {X 0,Y 608.472,Z 548.692,A -85,B 0,C 180,E1 -510.22,E2 -510.22} C_VEL
LIN {X 0,Y 608.478,Z 548.692,A -85,B 0,C 180,E1 -512.793,E2 -512.793} C_VEL
LIN {X 0,Y 608.449,Z 548.698,A -85,B 0,C 180,E1 -515.428,E2 -515.428} C_VEL
LIN {X 0,Y 608.47,Z 548.692,A -85,B 0,C 180,E1 -518.308,E2 -518.308} C_VEL
LIN {X 0,Y 608.476,Z 548.695,A -85,B 0,C 180,E1 -521.283,E2 -521.283} C_VEL
LIN {X 0,Y 608.461,Z 548.695,A -85,B 0,C 180,E1 -523.906,E2 -523.906} C_VEL
LIN {X 0,Y 608.459,Z 548.694,A -85,B 0,C 180,E1 -526.643,E2 -526.643} C_VEL
LIN {X 0,Y 608.465,Z 548.695,A -85,B 0,C 180,E1 -529.35,E2 -529.35} C_VEL
LIN {X 0,Y 608.477,Z 548.693,A -85,B 0,C 180,E1 -532.033,E2 -532.033} C_VEL
LIN {X 0,Y 608.462,Z 548.693,A -85,B 0,C 180,E1 -534.698,E2 -534.698} C_VEL
LIN {X 0,Y 608.482,Z 548.692,A -85,B 0,C 180,E1 -537.352,E2 -537.352} C_VEL
LIN {X 0,Y 608.48,Z 548.695,A -85,B 0,C 180,E1 -540,E2 -540} C_VEL
LIN {X 0,Y 608.482,Z 548.692,A -85,B 0,C 180,E1 -542.648,E2 -542.648} C_VEL
LIN {X 0,Y 608.462,Z 548.693,A -85,B 0,C 180,E1 -545.302,E2 -545.302} C_VEL
LIN {X 0,Y 608.482,Z 548.692,A -85,B 0,C 180,E1 -547.967,E2 -547.967} C_VEL
LIN {X 0,Y 608.458,Z 548.696,A -85,B 0,C 180,E1 -549.46,E2 -549.46} C_VEL
LIN {X 0,Y 607.776,Z 548.779,A -85,B 0,C 180,E1 -550.012,E2 -550.012} C_VEL
LIN {X 0,Y 604.922,Z 549.135,A -85,B 0,C 180,E1 -550.909,E2 -550.909} C_VEL
LIN {X 0,Y 602.523,Z 549.436,A -85,B 0,C 180,E1 -551.63,E2 -551.63} C_VEL
LIN {X 0,Y 601.495,Z 549.562,A -85,B 0,C 180,E1 -552.187,E2 -552.187} C_VEL
LIN {X 0,Y 601.412,Z 549.572,A -85,B 0,C 180,E1 -552.376,E2 -552.376} C_VEL
LIN {X 0,Y 601.434,Z 549.57,A -85,B 0,C 180,E1 -554.897,E2 -554.897} C_VEL
LIN {X 0,Y 601.433,Z 549.569,A -85,B 0,C 180,E1 -556.986,E2 -556.986} C_VEL
LIN {X 0,Y 601.405,Z 549.576,A -85,B 0,C 180,E1 -559.809,E2 -559.809} C_VEL
LIN {X 0,Y 601.414,Z 549.571,A -85,B 0,C 180,E1 -562.683,E2 -562.683} C_VEL
LIN {X 0,Y 601.401,Z 549.573,A -85,B 0,C 180,E1 -564.878,E2 -564.878} C_VEL
LIN {X 0,Y 601.423,Z 549.572,A -85,B 0,C 180,E1 -567.867,E2 -567.867} C_VEL
LIN {X 0,Y 601.43,Z 549.571,A -85,B 0,C 180,E1 -570.164,E2 -570.164} C_VEL
LIN {X 0,Y 601.42,Z 549.574,A -85,B 0,C 180,E1 -572.715,E2 -572.715} C_VEL
LIN {X 0,Y 601.415,Z 549.574,A -85,B 0,C 180,E1 -575.114,E2 -575.114} C_VEL
LIN {X 0,Y 601.436,Z 549.572,A -85,B 0,C 180,E1 -577.419,E2 -577.419} C_VEL
LIN {X 0,Y 601.412,Z 549.573,A -85,B 0,C 180,E1 -579.995,E2 -579.995} C_VEL
LIN {X 0,Y 601.41,Z 549.572,A -85,B 0,C 180,E1 -582.67,E2 -582.67} C_VEL
LIN {X 0,Y 601.427,Z 549.573,A -85,B 0,C 180,E1 -585.482,E2 -585.482} C_VEL
LIN {X 0,Y 601.428,Z 549.57,A -85,B 0,C 180,E1 -588.406,E2 -588.406} C_VEL
LIN {X 0,Y 601.437,Z 549.568,A -85,B 0,C 180,E1 -590.875,E2 -590.875} C_VEL
LIN {X 0,Y 601.402,Z 549.574,A -85,B 0,C 180,E1 -593.417,E2 -593.417} C_VEL
LIN {X 0,Y 601.432,Z 549.573,A -85,B 0,C 180,E1 -596.064,E2 -596.064} C_VEL
LIN {X 0,Y 601.444,Z 549.57,A -85,B 0,C 180,E1 -598.541,E2 -598.541} C_VEL
LIN {X 0,Y 601.427,Z 549.57,A -85,B 0,C 180,E1 -601.372,E2 -601.372} C_VEL
LIN {X 0,Y 601.407,Z 549.572,A -85,B 0,C 180,E1 -603.636,E2 -603.636} C_VEL
LIN {X 0,Y 601.423,Z 549.574,A -85,B 0,C 180,E1 -606.589,E2 -606.589} C_VEL
LIN {X 0,Y 601.427,Z 549.57,A -85,B 0,C 180,E1 -609.478,E2 -609.478} C_VEL
LIN {X 0,Y 601.4,Z 549.576,A -85,B 0,C 180,E1 -612.311,E2 -612.311} C_VEL
LIN {X 0,Y 601.42,Z 549.571,A -85,B 0,C 180,E1 -614.408,E2 -614.408} C_VEL
LIN {X 0,Y 601.42,Z 549.573,A -85,B 0,C 180,E1 -617.171,E2 -617.171} C_VEL
LIN {X 0,Y 601.438,Z 549.568,A -85,B 0,C 180,E1 -619.905,E2 -619.905} C_VEL
LIN {X 0,Y 601.442,Z 549.569,A -85,B 0,C 180,E1 -622.614,E2 -622.614} C_VEL
LIN {X 0,Y 601.427,Z 549.573,A -85,B 0,C 180,E1 -625.307,E2 -625.307} C_VEL
LIN {X 0,Y 601.435,Z 549.569,A -85,B 0,C 180,E1 -627.99,E2 -627.99} C_VEL
LIN {X 0,Y 601.443,Z 549.568,A -85,B 0,C 180,E1 -630.669,E2 -630.669} C_VEL
LIN {X 0,Y 601.46,Z 549.74,A -85,B 0,C 180,E1 -632.553,E2 -632.553} C_VEL
LIN {X 0,Y 601.539,Z 562.449,A -85,B 0,C 180,E1 -633.013,E2 -633.013} C_VEL
LIN {X 0,Y 601.519,Z 574.565,A -85,B 0,C 180,E1 -633.6,E2 -633.6} C_VEL
LIN {X 0,Y 601.474,Z 585.464,A -85,B 0,C 180,E1 -634.271,E2 -634.271} C_VEL
LIN {X 0,Y 601.455,Z 595.319,A -85,B 0,C 180,E1 -635.027,E2 -635.027} C_VEL
LIN {X 0,Y 601.401,Z 604.297,A -85,B 0,C 180,E1 -635.868,E2 -635.868} C_VEL
LIN {X 0,Y 601.383,Z 613.087,A -85,B 0,C 180,E1 -636.879,E2 -636.879} C_VEL
LIN {X 0,Y 601.361,Z 620.177,A -85,B 0,C 180,E1 -637.892,E2 -637.892} C_VEL
LIN {X 0,Y 601.348,Z 626.66,A -85,B 0,C 180,E1 -639.077,E2 -639.077} C_VEL
LIN {X 0,Y 601.337,Z 630.944,A -85,B 0,C 180,E1 -640.096,E2 -640.096} C_VEL
LIN {X 0,Y 601.351,Z 633.787,A -85,B 0,C 180,E1 -640.977,E2 -640.977} C_VEL
LIN {X 0,Y 601.341,Z 636.379,A -85,B 0,C 180,E1 -642.143,E2 -642.143} C_VEL
LIN {X 0,Y 601.324,Z 637.327,A -85,B 0,C 180,E1 -642.83,E2 -642.83} C_VEL
LIN {X 0,Y 601.345,Z 637.999,A -85,B 0,C 180,E1 -644.064,E2 -644.064} C_VEL
LIN {X 0,Y 601.314,Z 637.656,A -85,B 0,C 180,E1 -644.899,E2 -644.899} C_VEL
LIN {X 0,Y 601.325,Z 636.931,A -85,B 0,C 180,E1 -645.593,E2 -645.593} C_VEL
LIN {X 0,Y 601.322,Z 635.111,A -85,B 0,C 180,E1 -646.589,E2 -646.589} C_VEL
LIN {X 0,Y 601.326,Z 632.018,A -85,B 0,C 180,E1 -647.69,E2 -647.69} C_VEL
LIN {X 0,Y 601.348,Z 627.668,A -85,B 0,C 180,E1 -648.8,E2 -648.8} C_VEL
LIN {X 0,Y 601.369,Z 621.438,A -85,B 0,C 180,E1 -649.988,E2 -649.988} C_VEL
LIN {X 0,Y 601.397,Z 613.992,A -85,B 0,C 180,E1 -651.095,E2 -651.095} C_VEL
LIN {X 0,Y 601.386,Z 606.793,A -85,B 0,C 180,E1 -651.959,E2 -651.959} C_VEL
LIN {X 0,Y 601.418,Z 597.608,A -85,B 0,C 180,E1 -652.863,E2 -652.863} C_VEL
LIN {X 0,Y 601.461,Z 587.378,A -85,B 0,C 180,E1 -653.682,E2 -653.682} C_VEL
LIN {X 0,Y 601.498,Z 576.447,A -85,B 0,C 180,E1 -654.387,E2 -654.387} C_VEL
LIN {X 0,Y 601.528,Z 563.987,A -85,B 0,C 180,E1 -655.011,E2 -655.011} C_VEL
LIN {X 0,Y 601.546,Z 551.735,A -85,B 0,C 180,E1 -655.472,E2 -655.472} C_VEL
LIN {X 0,Y 601.421,Z 549.572,A -85,B 0,C 180,E1 -655.547,E2 -655.547} C_VEL
LIN {X 0,Y 601.418,Z 549.572,A -85,B 0,C 180,E1 -657.867,E2 -657.867} C_VEL
LIN {X 0,Y 601.444,Z 549.569,A -85,B 0,C 180,E1 -660.162,E2 -660.162} C_VEL
LIN {X 0,Y 601.423,Z 549.573,A -85,B 0,C 180,E1 -662.716,E2 -662.716} C_VEL
LIN {X 0,Y 601.39,Z 549.578,A -85,B 0,C 180,E1 -665.112,E2 -665.112} C_VEL
LIN {X 0,Y 601.432,Z 549.572,A -85,B 0,C 180,E1 -667.418,E2 -667.418} C_VEL
LIN {X 0,Y 601.413,Z 549.574,A -85,B 0,C 180,E1 -669.994,E2 -669.994} C_VEL
LIN {X 0,Y 601.455,Z 549.712,A -85,B 0,C 180,E1 -671.761,E2 -671.761} C_VEL
LIN {X 0,Y 601.506,Z 558.115,A -85,B 0,C 180,E1 -674.543,E2 -674.543} C_VEL
LIN {X 0,Y 601.485,Z 566.322,A -85,B 0,C 180,E1 -677.4,E2 -677.4} C_VEL
LIN {X 0,Y 601.434,Z 573.988,A -85,B 0,C 180,E1 -680.007,E2 -680.007} C_VEL
LIN {X 0,Y 601.432,Z 581.835,A -85,B 0,C 180,E1 -682.617,E2 -682.617} C_VEL
LIN {X 0,Y 601.413,Z 589.359,A -85,B 0,C 180,E1 -685.068,E2 -685.068} C_VEL
LIN {X 0,Y 601.372,Z 598.141,A -85,B 0,C 180,E1 -687.877,E2 -687.877} C_VEL
LIN {X 0,Y 601.373,Z 606.808,A -85,B 0,C 180,E1 -690.605,E2 -690.605} C_VEL
LIN {X 0,Y 601.35,Z 614.149,A -85,B 0,C 180,E1 -692.884,E2 -692.884} C_VEL
LIN {X 0,Y 601.374,Z 621.468,A -85,B 0,C 180,E1 -695.136,E2 -695.136} C_VEL
LIN {X 0,Y 601.617,Z 629.53,A -85,B 0,C 180,E1 -695.292,E2 -695.292} C_VEL
LIN {X 0,Y 601.557,Z 641.48,A -85,B 0,C 180,E1 -695.609,E2 -695.609} C_VEL
LIN {X 0,Y 601.537,Z 653.208,A -85,B 0,C 180,E1 -696.047,E2 -696.047} C_VEL
LIN {X 0,Y 601.489,Z 664.431,A -85,B 0,C 180,E1 -696.593,E2 -696.593} C_VEL
LIN {X 0,Y 601.49,Z 674.827,A -85,B 0,C 180,E1 -697.23,E2 -697.23} C_VEL
LIN {X 0,Y 601.431,Z 685.5,A -85,B 0,C 180,E1 -698.042,E2 -698.042} C_VEL
LIN {X 0,Y 601.428,Z 695.778,A -85,B 0,C 180,E1 -699.022,E2 -699.022} C_VEL
LIN {X 0,Y 601.392,Z 704.114,A -85,B 0,C 180,E1 -700.012,E2 -700.012} C_VEL
LIN {X 0,Y 601.393,Z 711.932,A -85,B 0,C 180,E1 -701.185,E2 -701.185} C_VEL
LIN {X 0,Y 601.348,Z 717.764,A -85,B 0,C 180,E1 -702.31,E2 -702.31} C_VEL
LIN {X 0,Y 601.327,Z 722.041,A -85,B 0,C 180,E1 -703.406,E2 -703.406} C_VEL
LIN {X 0,Y 601.33,Z 724.901,A -85,B 0,C 180,E1 -704.407,E2 -704.407} C_VEL
LIN {X 0,Y 601.313,Z 726.309,A -85,B 0,C 180,E1 -705.1,E2 -705.1} C_VEL
LIN {X 0,Y 601.339,Z 727.451,A -85,B 0,C 180,E1 -705.935,E2 -705.935} C_VEL
LIN {X 0,Y 601.322,Z 727.977,A -85,B 0,C 180,E1 -707.17,E2 -707.17} C_VEL
LIN {X 0,Y 601.339,Z 727.686,A -85,B 0,C 180,E1 -707.856,E2 -707.856} C_VEL
LIN {X 0,Y 601.348,Z 726.258,A -85,B 0,C 180,E1 -709.02,E2 -709.02} C_VEL
LIN {X 0,Y 601.327,Z 724.341,A -85,B 0,C 180,E1 -709.903,E2 -709.903} C_VEL
LIN {X 0,Y 601.346,Z 721.207,A -85,B 0,C 180,E1 -710.922,E2 -710.922} C_VEL
LIN {X 0,Y 601.348,Z 717.018,A -85,B 0,C 180,E1 -711.938,E2 -711.938} C_VEL
LIN {X 0,Y 601.371,Z 710.641,A -85,B 0,C 180,E1 -713.12,E2 -713.12} C_VEL
LIN {X 0,Y 601.385,Z 703.714,A -85,B 0,C 180,E1 -714.131,E2 -714.131} C_VEL
LIN {X 0,Y 601.402,Z 695.089,A -85,B 0,C 180,E1 -715.14,E2 -715.14} C_VEL
LIN {X 0,Y 601.421,Z 686.285,A -85,B 0,C 180,E1 -715.98,E2 -715.98} C_VEL
LIN {X 0,Y 601.47,Z 675.46,A -85,B 0,C 180,E1 -716.819,E2 -716.819} C_VEL
LIN {X 0,Y 601.501,Z 664.577,A -85,B 0,C 180,E1 -717.489,E2 -717.489} C_VEL
LIN {X 0,Y 601.506,Z 652.485,A -85,B 0,C 180,E1 -718.075,E2 -718.075} C_VEL
LIN {X 0,Y 601.592,Z 639.74,A -85,B 0,C 180,E1 -718.536,E2 -718.536} C_VEL
LIN {X 0,Y 601.582,Z 626.966,A -85,B 0,C 180,E1 -718.85,E2 -718.85} C_VEL
LIN {X 0,Y 601.364,Z 621.489,A -85,B 0,C 180,E1 -718.954,E2 -718.954} C_VEL
LIN {X 0,Y 601.395,Z 612.685,A -85,B 0,C 180,E1 -721.674,E2 -721.674} C_VEL
LIN {X 0,Y 601.393,Z 603.047,A -85,B 0,C 180,E1 -724.692,E2 -724.692} C_VEL
LIN {X 0,Y 601.395,Z 594.581,A -85,B 0,C 180,E1 -727.386,E2 -727.386} C_VEL
LIN {X 0,Y 601.414,Z 586.208,A -85,B 0,C 180,E1 -730.096,E2 -730.096} C_VEL
LIN {X 0,Y 601.464,Z 577.932,A -85,B 0,C 180,E1 -732.827,E2 -732.827} C_VEL
LIN {X 0,Y 601.465,Z 569.759,A -85,B 0,C 180,E1 -735.59,E2 -735.59} C_VEL
LIN {X 0,Y 601.467,Z 561.691,A -85,B 0,C 180,E1 -738.391,E2 -738.391} C_VEL
LIN {X 0,Y 601.443,Z 556.359,A -85,B 0,C 180,E1 -740.165,E2 -740.165} C_VEL
LIN {X 0,Y 601.407,Z 549.574,A -85,B 0,C 180,E1 -742.138,E2 -742.138} C_VEL
LIN {X 0,Y 601.405,Z 549.576,A -85,B 0,C 180,E1 -744.879,E2 -744.879} C_VEL
LIN {X 0,Y 601.423,Z 549.572,A -85,B 0,C 180,E1 -747.868,E2 -747.868} C_VEL
LIN {X 0,Y 601.444,Z 549.571,A -85,B 0,C 180,E1 -750.163,E2 -750.163} C_VEL
LIN {X 0,Y 601.427,Z 549.571,A -85,B 0,C 180,E1 -752.718,E2 -752.718} C_VEL
LIN {X 0,Y 601.417,Z 549.573,A -85,B 0,C 180,E1 -755.117,E2 -755.117} C_VEL
LIN {X 0,Y 601.432,Z 549.573,A -85,B 0,C 180,E1 -757.42,E2 -757.42} C_VEL
LIN {X 0,Y 601.41,Z 549.573,A -85,B 0,C 180,E1 -759.995,E2 -759.995} C_VEL
LIN {X 0,Y 601.409,Z 549.575,A -85,B 0,C 180,E1 -762.671,E2 -762.671} C_VEL
LIN {X 0,Y 601.422,Z 549.572,A -85,B 0,C 180,E1 -765.483,E2 -765.483} C_VEL
LIN {X 0,Y 601.423,Z 549.571,A -85,B 0,C 180,E1 -768.407,E2 -768.407} C_VEL
LIN {X 0,Y 601.436,Z 549.572,A -85,B 0,C 180,E1 -770.877,E2 -770.877} C_VEL
LIN {X 0,Y 601.443,Z 549.57,A -85,B 0,C 180,E1 -773.735,E2 -773.735} C_VEL
LIN {X 0,Y 601.433,Z 549.584,A -85,B 0,C 180,E1 -774.114,E2 -774.114} C_VEL
LIN {X 0,Y 601.74,Z 555.575,A -85,B 0,C 180,E1 -775.295,E2 -775.295} C_VEL
LIN {X 0,Y 601.804,Z 567.032,A -85,B 0,C 180,E1 -777.508,E2 -777.508} C_VEL
LIN {X 0,Y 601.714,Z 580.782,A -85,B 0,C 180,E1 -780.239,E2 -780.239} C_VEL
LIN {X 0,Y 601.687,Z 594.532,A -85,B 0,C 180,E1 -782.901,E2 -782.901} C_VEL
LIN {X 0,Y 601.6,Z 609.213,A -85,B 0,C 180,E1 -785.674,E2 -785.674} C_VEL
LIN {X 0,Y 601.55,Z 623.996,A -85,B 0,C 180,E1 -788.407,E2 -788.407} C_VEL
LIN {X 0,Y 601.484,Z 640.407,A -85,B 0,C 180,E1 -791.383,E2 -791.383} C_VEL
LIN {X 0,Y 601.476,Z 655.424,A -85,B 0,C 180,E1 -794.063,E2 -794.063} C_VEL
LIN {X 0,Y 601.403,Z 671.138,A -85,B 0,C 180,E1 -796.829,E2 -796.829} C_VEL
LIN {X 0,Y 601.411,Z 678.139,A -85,B 0,C 180,E1 -798.051,E2 -798.051} C_VEL
LIN {X 0,Y 601.589,Z 690.47,A -85,B 0,C 180,E1 -798.268,E2 -798.268} C_VEL
LIN {X 0,Y 601.56,Z 703.286,A -85,B 0,C 180,E1 -798.624,E2 -798.624} C_VEL
LIN {X 0,Y 601.515,Z 715.863,A -85,B 0,C 180,E1 -799.115,E2 -799.115} C_VEL
LIN {X 0,Y 601.484,Z 727.768,A -85,B 0,C 180,E1 -799.737,E2 -799.737} C_VEL
LIN {X 0,Y 601.462,Z 739.262,A -85,B 0,C 180,E1 -800.501,E2 -800.501} C_VEL
LIN {X 0,Y 601.436,Z 748.544,A -85,B 0,C 180,E1 -801.263,E2 -801.263} C_VEL
LIN {X 0,Y 601.4,Z 756.995,A -85,B 0,C 180,E1 -802.108,E2 -802.108} C_VEL
LIN {X 0,Y 601.381,Z 765.24,A -85,B 0,C 180,E1 -803.121,E2 -803.121} C_VEL
LIN {X 0,Y 601.372,Z 771.881,A -85,B 0,C 180,E1 -804.131,E2 -804.131} C_VEL
LIN {X 0,Y 601.337,Z 777.953,A -85,B 0,C 180,E1 -805.308,E2 -805.308} C_VEL
LIN {X 0,Y 601.367,Z 781.898,A -85,B 0,C 180,E1 -806.315,E2 -806.315} C_VEL
LIN {X 0,Y 601.325,Z 784.811,A -85,B 0,C 180,E1 -807.321,E2 -807.321} C_VEL
LIN {X 0,Y 601.34,Z 786.203,A -85,B 0,C 180,E1 -807.991,E2 -807.991} C_VEL
LIN {X 0,Y 601.339,Z 787.784,A -85,B 0,C 180,E1 -809.331,E2 -809.331} C_VEL
LIN {X 0,Y 601.335,Z 788,A -85,B 0,C 180,E1 -810.001,E2 -810.001} C_VEL
LIN {X 0,Y 601.348,Z 787.183,A -85,B 0,C 180,E1 -811.34,E2 -811.34} C_VEL
LIN {X 0,Y 601.34,Z 786.201,A -85,B 0,C 180,E1 -812.01,E2 -812.01} C_VEL
LIN {X 0,Y 601.325,Z 784.808,A -85,B 0,C 180,E1 -812.68,E2 -812.68} C_VEL
LIN {X 0,Y 601.367,Z 781.894,A -85,B 0,C 180,E1 -813.686,E2 -813.686} C_VEL
LIN {X 0,Y 601.337,Z 777.947,A -85,B 0,C 180,E1 -814.693,E2 -814.693} C_VEL
LIN {X 0,Y 601.372,Z 771.873,A -85,B 0,C 180,E1 -815.87,E2 -815.87} C_VEL
LIN {X 0,Y 601.382,Z 765.231,A -85,B 0,C 180,E1 -816.88,E2 -816.88} C_VEL
LIN {X 0,Y 601.4,Z 756.984,A -85,B 0,C 180,E1 -817.893,E2 -817.893} C_VEL
LIN {X 0,Y 601.436,Z 748.53,A -85,B 0,C 180,E1 -818.738,E2 -818.738} C_VEL
LIN {X 0,Y 601.448,Z 738.084,A -85,B 0,C 180,E1 -819.586,E2 -819.586} C_VEL
LIN {X 0,Y 601.484,Z 727.748,A -85,B 0,C 180,E1 -820.265,E2 -820.265} C_VEL
LIN {X 0,Y 601.536,Z 715.877,A -85,B 0,C 180,E1 -820.884,E2 -820.884} C_VEL
LIN {X 0,Y 601.561,Z 703.255,A -85,B 0,C 180,E1 -821.377,E2 -821.377} C_VEL
LIN {X 0,Y 601.59,Z 690.415,A -85,B 0,C 180,E1 -821.733,E2 -821.733} C_VEL
LIN {X 0,Y 601.412,Z 678.153,A -85,B 0,C 180,E1 -821.951,E2 -821.951} C_VEL
LIN {X 0,Y 601.436,Z 661.402,A -85,B 0,C 180,E1 -824.897,E2 -824.897} C_VEL
LIN {X 0,Y 601.485,Z 645.751,A -85,B 0,C 180,E1 -827.686,E2 -827.686} C_VEL
LIN {X 0,Y 601.507,Z 630.099,A -85,B 0,C 180,E1 -830.52,E2 -830.52} C_VEL
LIN {X 0,Y 601.586,Z 616.405,A -85,B 0,C 180,E1 -833.04,E2 -833.04} C_VEL
LIN {X 0,Y 601.654,Z 600.217,A -85,B 0,C 180,E1 -836.082,E2 -836.082} C_VEL
LIN {X 0,Y 601.714,Z 584.792,A -85,B 0,C 180,E1 -839.055,E2 -839.055} C_VEL
LIN {X 0,Y 601.783,Z 571.407,A -85,B 0,C 180,E1 -841.705,E2 -841.705} C_VEL
LIN {X 0,Y 601.761,Z 561.716,A -85,B 0,C 180,E1 -843.638,E2 -843.638} C_VEL
LIN {X 0,Y 601.664,Z 550.893,A -85,B 0,C 180,E1 -845.736,E2 -845.736} C_VEL
LIN {X 0,Y 601.421,Z 549.574,A -85,B 0,C 180,E1 -846.022,E2 -846.022} C_VEL
LIN {X 0,Y 601.438,Z 549.571,A -85,B 0,C 180,E1 -848.471,E2 -848.471} C_VEL
LIN {X 0,Y 601.42,Z 549.574,A -85,B 0,C 180,E1 -850.874,E2 -850.874} C_VEL
LIN {X 0,Y 601.434,Z 549.57,A -85,B 0,C 180,E1 -853.586,E2 -853.586} C_VEL
LIN {X 0,Y 601.455,Z 549.567,A -85,B 0,C 180,E1 -856.425,E2 -856.425} C_VEL
LIN {X 0,Y 601.414,Z 549.572,A -85,B 0,C 180,E1 -859.427,E2 -859.427} C_VEL
LIN {X 0,Y 601.415,Z 549.572,A -85,B 0,C 180,E1 -861.731,E2 -861.731} C_VEL
LIN {X 0,Y 601.412,Z 549.572,A -85,B 0,C 180,E1 -864.247,E2 -864.247} C_VEL
LIN {X 0,Y 601.42,Z 549.571,A -85,B 0,C 180,E1 -866.686,E2 -866.686} C_VEL
LIN {X 0,Y 601.415,Z 549.571,A -85,B 0,C 180,E1 -869.057,E2 -869.057} C_VEL
LIN {X 0,Y 601.436,Z 549.568,A -85,B 0,C 180,E1 -871.373,E2 -871.373} C_VEL
LIN {X 0,Y 601.42,Z 549.573,A -85,B 0,C 180,E1 -874.132,E2 -874.132} C_VEL
LIN {X 0,Y 601.422,Z 549.574,A -85,B 0,C 180,E1 -876.589,E2 -876.589} C_VEL
LIN {X 0,Y 601.436,Z 549.569,A -85,B 0,C 180,E1 -879.478,E2 -879.478} C_VEL
LIN {X 0,Y 601.394,Z 549.576,A -85,B 0,C 180,E1 -882.311,E2 -882.311} C_VEL
LIN {X 0,Y 601.417,Z 549.571,A -85,B 0,C 180,E1 -884.409,E2 -884.409} C_VEL
LIN {X 0,Y 601.422,Z 549.574,A -85,B 0,C 180,E1 -887.172,E2 -887.172} C_VEL
LIN {X 0,Y 601.431,Z 549.57,A -85,B 0,C 180,E1 -889.905,E2 -889.905} C_VEL
LIN {X 0,Y 601.444,Z 549.568,A -85,B 0,C 180,E1 -892.615,E2 -892.615} C_VEL
LIN {X 0,Y 601.433,Z 549.573,A -85,B 0,C 180,E1 -895.308,E2 -895.308} C_VEL
LIN {X 0,Y 601.419,Z 549.572,A -85,B 0,C 180,E1 -897.991,E2 -897.991} C_VEL
LIN {X 0,Y 601.452,Z 549.567,A -85,B 0,C 180,E1 -900.669,E2 -900.669} C_VEL
LIN {X 0,Y 601.428,Z 549.572,A -85,B 0,C 180,E1 -903.349,E2 -903.349} C_VEL
LIN {X 0,Y 601.42,Z 549.572,A -85,B 0,C 180,E1 -906.037,E2 -906.037} C_VEL
LIN {X 0,Y 601.419,Z 549.571,A -85,B 0,C 180,E1 -908.738,E2 -908.738} C_VEL
LIN {X 0,Y 601.424,Z 549.571,A -85,B 0,C 180,E1 -911.458,E2 -911.458} C_VEL
LIN {X 0,Y 601.412,Z 549.572,A -85,B 0,C 180,E1 -912.376,E2 -912.376} C_VEL
LIN {X 0,Y 600.748,Z 549.657,A -85,B 0,C 180,E1 -912.935,E2 -912.935} C_VEL
LIN {X 0,Y 597.898,Z 550.013,A -85,B 0,C 180,E1 -913.843,E2 -913.843} C_VEL
LIN {X 0,Y 595.488,Z 550.313,A -85,B 0,C 180,E1 -914.573,E2 -914.573} C_VEL
LIN {X 0,Y 594.452,Z 550.442,A -85,B 0,C 180,E1 -915.136,E2 -915.136} C_VEL
LIN {X 0,Y 594.366,Z 550.45,A -85,B 0,C 180,E1 -915.327,E2 -915.327} C_VEL
LIN {X 0,Y 594.389,Z 550.447,A -85,B 0,C 180,E1 -917.193,E2 -917.193} C_VEL
LIN {X 0,Y 594.375,Z 550.45,A -85,B 0,C 180,E1 -920.053,E2 -920.053} C_VEL
LIN {X 0,Y 594.366,Z 550.45,A -85,B 0,C 180,E1 -922.967,E2 -922.967} C_VEL
LIN {X 0,Y 594.378,Z 550.448,A -85,B 0,C 180,E1 -925.193,E2 -925.193} C_VEL
LIN {X 0,Y 594.388,Z 550.446,A -85,B 0,C 180,E1 -927.526,E2 -927.526} C_VEL
LIN {X 0,Y 594.387,Z 550.45,A -85,B 0,C 180,E1 -930.328,E2 -930.328} C_VEL
LIN {X 0,Y 594.379,Z 550.449,A -85,B 0,C 180,E1 -932.95,E2 -932.95} C_VEL
LIN {X 0,Y 594.385,Z 550.447,A -85,B 0,C 180,E1 -935.406,E2 -935.406} C_VEL
LIN {X 0,Y 594.386,Z 550.447,A -85,B 0,C 180,E1 -937.94,E2 -937.94} C_VEL
LIN {X 0,Y 594.378,Z 550.451,A -85,B 0,C 180,E1 -940.822,E2 -940.822} C_VEL
LIN {X 0,Y 594.384,Z 550.447,A -85,B 0,C 180,E1 -943.841,E2 -943.841} C_VEL
LIN {X 0,Y 594.381,Z 550.451,A -85,B 0,C 180,E1 -946.701,E2 -946.701} C_VEL
LIN {X 0,Y 594.376,Z 550.448,A -85,B 0,C 180,E1 -949.433,E2 -949.433} C_VEL
LIN {X 0,Y 594.392,Z 550.448,A -85,B 0,C 180,E1 -952.391,E2 -952.391} C_VEL
LIN {X 0,Y 594.379,Z 550.447,A -85,B 0,C 180,E1 -955.42,E2 -955.42} C_VEL
LIN {X 0,Y 594.395,Z 550.449,A -85,B 0,C 180,E1 -958.354,E2 -958.354} C_VEL
LIN {X 0,Y 594.382,Z 550.448,A -85,B 0,C 180,E1 -961.042,E2 -961.042} C_VEL
LIN {X 0,Y 594.391,Z 550.447,A -85,B 0,C 180,E1 -963.976,E2 -963.976} C_VEL
LIN {X 0,Y 594.394,Z 550.447,A -85,B 0,C 180,E1 -966.296,E2 -966.296} C_VEL
LIN {X 0,Y 594.399,Z 550.446,A -85,B 0,C 180,E1 -969.224,E2 -969.224} C_VEL
LIN {X 0,Y 594.357,Z 550.451,A -85,B 0,C 180,E1 -972.095,E2 -972.095} C_VEL
LIN {X 0,Y 594.372,Z 550.448,A -85,B 0,C 180,E1 -974.219,E2 -974.219} C_VEL
LIN {X 0,Y 594.367,Z 550.452,A -85,B 0,C 180,E1 -977.016,E2 -977.016} C_VEL
LIN {X 0,Y 594.397,Z 550.446,A -85,B 0,C 180,E1 -979.784,E2 -979.784} C_VEL
LIN {X 0,Y 594.395,Z 550.446,A -85,B 0,C 180,E1 -982.526,E2 -982.526} C_VEL
LIN {X 0,Y 594.396,Z 550.449,A -85,B 0,C 180,E1 -985.252,E2 -985.252} C_VEL
LIN {X 0,Y 594.404,Z 550.445,A -85,B 0,C 180,E1 -987.967,E2 -987.967} C_VEL
LIN {X 0,Y 594.415,Z 550.444,A -85,B 0,C 180,E1 -990.677,E2 -990.677} C_VEL
LIN {X 0,Y 594.4,Z 550.448,A -85,B 0,C 180,E1 -992.435,E2 -992.435} C_VEL
LIN {X 0,Y 594.555,Z 562.367,A -85,B 0,C 180,E1 -992.879,E2 -992.879} C_VEL
LIN {X 0,Y 594.515,Z 574.516,A -85,B 0,C 180,E1 -993.473,E2 -993.473} C_VEL
LIN {X 0,Y 594.456,Z 585.426,A -85,B 0,C 180,E1 -994.152,E2 -994.152} C_VEL
LIN {X 0,Y 594.417,Z 595.285,A -85,B 0,C 180,E1 -994.917,E2 -994.917} C_VEL
LIN {X 0,Y 594.344,Z 604.268,A -85,B 0,C 180,E1 -995.768,E2 -995.768} C_VEL
LIN {X 0,Y 594.346,Z 611.936,A -85,B 0,C 180,E1 -996.649,E2 -996.649} C_VEL
LIN {X 0,Y 594.298,Z 619.049,A -85,B 0,C 180,E1 -997.645,E2 -997.645} C_VEL
LIN {X 0,Y 594.297,Z 624.041,A -85,B 0,C 180,E1 -998.5,E2 -998.5} C_VEL
LIN {X 0,Y 594.268,Z 628.913,A -85,B 0,C 180,E1 -999.53,E2 -999.53} C_VEL
LIN {X 0,Y 594.281,Z 632.658,A -85,B 0,C 180,E1 -1000.562,E2 -1000.562} C_VEL
LIN {X 0,Y 594.231,Z 635.38,A -85,B 0,C 180,E1 -1001.598,E2 -1001.598} C_VEL
LIN {X 0,Y 594.238,Z 636.656,A -85,B 0,C 180,E1 -1002.291,E2 -1002.291} C_VEL
LIN {X 0,Y 594.242,Z 637.516,A -85,B 0,C 180,E1 -1002.985,E2 -1002.985} C_VEL
LIN {X 0,Y 594.256,Z 637.988,A -85,B 0,C 180,E1 -1004.124,E2 -1004.124} C_VEL
LIN {X 0,Y 594.209,Z 637.536,A -85,B 0,C 180,E1 -1005.081,E2 -1005.081} C_VEL
LIN {X 0,Y 594.251,Z 636.681,A -85,B 0,C 180,E1 -1005.783,E2 -1005.783} C_VEL
LIN {X 0,Y 594.236,Z 634.991,A -85,B 0,C 180,E1 -1006.669,E2 -1006.669} C_VEL
LIN {X 0,Y 594.24,Z 631.432,A -85,B 0,C 180,E1 -1007.908,E2 -1007.908} C_VEL
LIN {X 0,Y 594.278,Z 626.637,A -85,B 0,C 180,E1 -1009.078,E2 -1009.078} C_VEL
LIN {X 0,Y 594.298,Z 620.39,A -85,B 0,C 180,E1 -1010.236,E2 -1010.236} C_VEL
LIN {X 0,Y 594.317,Z 612.772,A -85,B 0,C 180,E1 -1011.336,E2 -1011.336} C_VEL
LIN {X 0,Y 594.37,Z 605.118,A -85,B 0,C 180,E1 -1012.232,E2 -1012.232} C_VEL
LIN {X 0,Y 594.387,Z 595.559,A -85,B 0,C 180,E1 -1013.149,E2 -1013.149} C_VEL
LIN {X 0,Y 594.448,Z 584.829,A -85,B 0,C 180,E1 -1013.978,E2 -1013.978} C_VEL
LIN {X 0,Y 594.526,Z 573.333,A -85,B 0,C 180,E1 -1014.682,E2 -1014.682} C_VEL
LIN {X 0,Y 594.53,Z 561.878,A -85,B 0,C 180,E1 -1015.232,E2 -1015.232} C_VEL
LIN {X 0,Y 594.486,Z 551.09,A -85,B 0,C 180,E1 -1015.63,E2 -1015.63} C_VEL
LIN {X 0,Y 594.375,Z 550.451,A -85,B 0,C 180,E1 -1015.661,E2 -1015.661} C_VEL
LIN {X 0,Y 594.38,Z 550.451,A -85,B 0,C 180,E1 -1018.226,E2 -1018.226} C_VEL
LIN {X 0,Y 594.392,Z 550.449,A -85,B 0,C 180,E1 -1020.558,E2 -1020.558} C_VEL
LIN {X 0,Y 594.375,Z 550.45,A -85,B 0,C 180,E1 -1022.949,E2 -1022.949} C_VEL
LIN {X 0,Y 594.349,Z 550.452,A -85,B 0,C 180,E1 -1025.408,E2 -1025.408} C_VEL
LIN {X 0,Y 594.386,Z 550.447,A -85,B 0,C 180,E1 -1027.94,E2 -1027.94} C_VEL
LIN {X 0,Y 594.388,Z 550.449,A -85,B 0,C 180,E1 -1030.824,E2 -1030.824} C_VEL
LIN {X 0,Y 594.387,Z 550.448,A -85,B 0,C 180,E1 -1031.662,E2 -1031.662} C_VEL
LIN {X 0,Y 594.451,Z 557.009,A -85,B 0,C 180,E1 -1033.848,E2 -1033.848} C_VEL
LIN {X 0,Y 594.479,Z 565.454,A -85,B 0,C 180,E1 -1036.711,E2 -1036.711} C_VEL
LIN {X 0,Y 594.419,Z 573.332,A -85,B 0,C 180,E1 -1039.438,E2 -1039.438} C_VEL
LIN {X 0,Y 594.401,Z 581.094,A -85,B 0,C 180,E1 -1042.061,E2 -1042.061} C_VEL
LIN {X 0,Y 594.356,Z 588.995,A -85,B 0,C 180,E1 -1044.674,E2 -1044.674} C_VEL
LIN {X 0,Y 594.343,Z 597.618,A -85,B 0,C 180,E1 -1047.473,E2 -1047.473} C_VEL
LIN {X 0,Y 594.318,Z 606.23,A -85,B 0,C 180,E1 -1050.221,E2 -1050.221} C_VEL
LIN {X 0,Y 594.28,Z 614.8,A -85,B 0,C 180,E1 -1052.916,E2 -1052.916} C_VEL
LIN {X 0,Y 594.294,Z 621.465,A -85,B 0,C 180,E1 -1054.991,E2 -1054.991} C_VEL
LIN {X 0,Y 594.665,Z 626.966,A -85,B 0,C 180,E1 -1055.101,E2 -1055.101} C_VEL
LIN {X 0,Y 594.615,Z 639.985,A -85,B 0,C 180,E1 -1055.425,E2 -1055.425} C_VEL
LIN {X 0,Y 594.566,Z 652.535,A -85,B 0,C 180,E1 -1055.887,E2 -1055.887} C_VEL
LIN {X 0,Y 594.495,Z 663.055,A -85,B 0,C 180,E1 -1056.393,E2 -1056.393} C_VEL
LIN {X 0,Y 594.448,Z 673.699,A -85,B 0,C 180,E1 -1057.036,E2 -1057.036} C_VEL
LIN {X 0,Y 594.421,Z 684.646,A -85,B 0,C 180,E1 -1057.861,E2 -1057.861} C_VEL
LIN {X 0,Y 594.355,Z 693.288,A -85,B 0,C 180,E1 -1058.664,E2 -1058.664} C_VEL
LIN {X 0,Y 594.311,Z 701.43,A -85,B 0,C 180,E1 -1059.583,E2 -1059.583} C_VEL
LIN {X 0,Y 594.316,Z 709.189,A -85,B 0,C 180,E1 -1060.664,E2 -1060.664} C_VEL
LIN {X 0,Y 594.272,Z 715.302,A -85,B 0,C 180,E1 -1061.736,E2 -1061.736} C_VEL
LIN {X 0,Y 594.258,Z 720.047,A -85,B 0,C 180,E1 -1062.803,E2 -1062.803} C_VEL
LIN {X 0,Y 594.246,Z 723.587,A -85,B 0,C 180,E1 -1063.864,E2 -1063.864} C_VEL
LIN {X 0,Y 594.226,Z 726.047,A -85,B 0,C 180,E1 -1064.919,E2 -1064.919} C_VEL
LIN {X 0,Y 594.25,Z 727.396,A -85,B 0,C 180,E1 -1065.875,E2 -1065.875} C_VEL
LIN {X 0,Y 594.24,Z 727.998,A -85,B 0,C 180,E1 -1067.014,E2 -1067.014} C_VEL
LIN {X 0,Y 594.236,Z 727.794,A -85,B 0,C 180,E1 -1067.709,E2 -1067.709} C_VEL
LIN {X 0,Y 594.248,Z 726.18,A -85,B 0,C 180,E1 -1069.093,E2 -1069.093} C_VEL
LIN {X 0,Y 594.23,Z 724.744,A -85,B 0,C 180,E1 -1069.782,E2 -1069.782} C_VEL
LIN {X 0,Y 594.261,Z 721.76,A -85,B 0,C 180,E1 -1070.813,E2 -1070.813} C_VEL
LIN {X 0,Y 594.276,Z 717.737,A -85,B 0,C 180,E1 -1071.842,E2 -1071.842} C_VEL
LIN {X 0,Y 594.297,Z 711.562,A -85,B 0,C 180,E1 -1073.038,E2 -1073.038} C_VEL
LIN {X 0,Y 594.322,Z 704.843,A -85,B 0,C 180,E1 -1074.061,E2 -1074.061} C_VEL
LIN {X 0,Y 594.345,Z 696.522,A -85,B 0,C 180,E1 -1075.082,E2 -1075.082} C_VEL
LIN {X 0,Y 594.386,Z 688.029,A -85,B 0,C 180,E1 -1075.932,E2 -1075.932} C_VEL
LIN {X 0,Y 594.465,Z 677.592,A -85,B 0,C 180,E1 -1076.781,E2 -1076.781} C_VEL
LIN {X 0,Y 594.484,Z 667.305,A -85,B 0,C 180,E1 -1077.459,E2 -1077.459} C_VEL
LIN {X 0,Y 594.518,Z 655.985,A -85,B 0,C 180,E1 -1078.053,E2 -1078.053} C_VEL
LIN {X 0,Y 594.588,Z 644.389,A -85,B 0,C 180,E1 -1078.519,E2 -1078.519} C_VEL
LIN {X 0,Y 594.644,Z 632.037,A -85,B 0,C 180,E1 -1078.879,E2 -1078.879} C_VEL
LIN {X 0,Y 594.458,Z 622.743,A -85,B 0,C 180,E1 -1079.069,E2 -1079.069} C_VEL
LIN {X 0,Y 594.291,Z 621.447,A -85,B 0,C 180,E1 -1079.111,E2 -1079.111} C_VEL
LIN {X 0,Y 594.339,Z 613.186,A -85,B 0,C 180,E1 -1081.694,E2 -1081.694} C_VEL
LIN {X 0,Y 594.332,Z 603.55,A -85,B 0,C 180,E1 -1084.748,E2 -1084.748} C_VEL
LIN {X 0,Y 594.359,Z 595.084,A -85,B 0,C 180,E1 -1087.474,E2 -1087.474} C_VEL
LIN {X 0,Y 594.37,Z 586.716,A -85,B 0,C 180,E1 -1090.217,E2 -1090.217} C_VEL
LIN {X 0,Y 594.422,Z 578.445,A -85,B 0,C 180,E1 -1092.982,E2 -1092.982} C_VEL
LIN {X 0,Y 594.44,Z 570.277,A -85,B 0,C 180,E1 -1095.779,E2 -1095.779} C_VEL
LIN {X 0,Y 594.479,Z 563.215,A -85,B 0,C 180,E1 -1098.258,E2 -1098.258} C_VEL
LIN {X 0,Y 594.345,Z 553.695,A -85,B 0,C 180,E1 -1101.171,E2 -1101.171} C_VEL
LIN {X 0,Y 594.34,Z 550.454,A -85,B 0,C 180,E1 -1102.143,E2 -1102.143} C_VEL
LIN {X 0,Y 594.383,Z 550.448,A -85,B 0,C 180,E1 -1104.447,E2 -1104.447} C_VEL
LIN {X 0,Y 594.387,Z 550.448,A -85,B 0,C 180,E1 -1106.7,E2 -1106.7} C_VEL
LIN {X 0,Y 594.381,Z 550.45,A -85,B 0,C 180,E1 -1108.999,E2 -1108.999} C_VEL
LIN {X 0,Y 594.391,Z 550.447,A -85,B 0,C 180,E1 -1111.647,E2 -1111.647} C_VEL
LIN {X 0,Y 594.396,Z 550.447,A -85,B 0,C 180,E1 -1114.579,E2 -1114.579} C_VEL
LIN {X 0,Y 594.383,Z 550.448,A -85,B 0,C 180,E1 -1117.087,E2 -1117.087} C_VEL
LIN {X 0,Y 594.375,Z 550.449,A -85,B 0,C 180,E1 -1119.776,E2 -1119.776} C_VEL
LIN {X 0,Y 594.366,Z 550.451,A -85,B 0,C 180,E1 -1122.376,E2 -1122.376} C_VEL
LIN {X 0,Y 594.359,Z 550.451,A -85,B 0,C 180,E1 -1125.192,E2 -1125.192} C_VEL
LIN {X 0,Y 594.369,Z 550.452,A -85,B 0,C 180,E1 -1127.626,E2 -1127.626} C_VEL
LIN {X 0,Y 594.39,Z 550.447,A -85,B 0,C 180,E1 -1130.322,E2 -1130.322} C_VEL
LIN {X 0,Y 594.386,Z 550.451,A -85,B 0,C 180,E1 -1132.915,E2 -1132.915} C_VEL
LIN {X 0,Y 594.42,Z 550.486,A -85,B 0,C 180,E1 -1133.919,E2 -1133.919} C_VEL
LIN {X 0,Y 594.819,Z 555.012,A -85,B 0,C 180,E1 -1134.832,E2 -1134.832} C_VEL
LIN {X 0,Y 594.931,Z 568.861,A -85,B 0,C 180,E1 -1137.488,E2 -1137.488} C_VEL
LIN {X 0,Y 594.838,Z 582.747,A -85,B 0,C 180,E1 -1140.25,E2 -1140.25} C_VEL
LIN {X 0,Y 594.757,Z 596.496,A -85,B 0,C 180,E1 -1142.94,E2 -1142.94} C_VEL
LIN {X 0,Y 594.645,Z 612.21,A -85,B 0,C 180,E1 -1145.937,E2 -1145.937} C_VEL
LIN {X 0,Y 594.556,Z 625.96,A -85,B 0,C 180,E1 -1148.505,E2 -1148.505} C_VEL
LIN {X 0,Y 594.491,Z 641.674,A -85,B 0,C 180,E1 -1151.387,E2 -1151.387} C_VEL
LIN {X 0,Y 594.431,Z 657.388,A -85,B 0,C 180,E1 -1154.222,E2 -1154.222} C_VEL
LIN {X 0,Y 594.343,Z 673.102,A -85,B 0,C 180,E1 -1157.017,E2 -1157.017} C_VEL
LIN {X 0,Y 594.356,Z 678.139,A -85,B 0,C 180,E1 -1157.907,E2 -1157.907} C_VEL
LIN {X 0,Y 594.674,Z 686.269,A -85,B 0,C 180,E1 -1158.043,E2 -1158.043} C_VEL
LIN {X 0,Y 594.611,Z 699.522,A -85,B 0,C 180,E1 -1158.366,E2 -1158.366} C_VEL
LIN {X 0,Y 594.571,Z 711.932,A -85,B 0,C 180,E1 -1158.814,E2 -1158.814} C_VEL
LIN {X 0,Y 594.507,Z 723.222,A -85,B 0,C 180,E1 -1159.356,E2 -1159.356} C_VEL
LIN {X 0,Y 594.46,Z 734.487,A -85,B 0,C 180,E1 -1160.044,E2 -1160.044} C_VEL
LIN {X 0,Y 594.406,Z 744.655,A -85,B 0,C 180,E1 -1160.816,E2 -1160.816} C_VEL
LIN {X 0,Y 594.372,Z 753.794,A -85,B 0,C 180,E1 -1161.672,E2 -1161.672} C_VEL
LIN {X 0,Y 594.316,Z 762.696,A -85,B 0,C 180,E1 -1162.697,E2 -1162.697} C_VEL
LIN {X 0,Y 594.281,Z 769.171,A -85,B 0,C 180,E1 -1163.615,E2 -1163.615} C_VEL
LIN {X 0,Y 594.289,Z 774.684,A -85,B 0,C 180,E1 -1164.572,E2 -1164.572} C_VEL
LIN {X 0,Y 594.27,Z 779.374,A -85,B 0,C 180,E1 -1165.592,E2 -1165.592} C_VEL
LIN {X 0,Y 594.268,Z 782.958,A -85,B 0,C 180,E1 -1166.611,E2 -1166.611} C_VEL
LIN {X 0,Y 594.226,Z 784.81,A -85,B 0,C 180,E1 -1167.289,E2 -1167.289} C_VEL
LIN {X 0,Y 594.239,Z 786.203,A -85,B 0,C 180,E1 -1167.967,E2 -1167.967} C_VEL
LIN {X 0,Y 594.239,Z 787.784,A -85,B 0,C 180,E1 -1169.323,E2 -1169.323} C_VEL
LIN {X 0,Y 594.236,Z 788,A -85,B 0,C 180,E1 -1170.001,E2 -1170.001} C_VEL
LIN {X 0,Y 594.247,Z 787.184,A -85,B 0,C 180,E1 -1171.356,E2 -1171.356} C_VEL
LIN {X 0,Y 594.239,Z 786.201,A -85,B 0,C 180,E1 -1172.034,E2 -1172.034} C_VEL
LIN {X 0,Y 594.226,Z 784.808,A -85,B 0,C 180,E1 -1172.712,E2 -1172.712} C_VEL
LIN {X 0,Y 594.288,Z 781.894,A -85,B 0,C 180,E1 -1173.73,E2 -1173.73} C_VEL
LIN {X 0,Y 594.242,Z 777.947,A -85,B 0,C 180,E1 -1174.749,E2 -1174.749} C_VEL
LIN {X 0,Y 594.304,Z 771.874,A -85,B 0,C 180,E1 -1175.94,E2 -1175.94} C_VEL
LIN {X 0,Y 594.309,Z 765.232,A -85,B 0,C 180,E1 -1176.963,E2 -1176.963} C_VEL
LIN {X 0,Y 594.359,Z 756.985,A -85,B 0,C 180,E1 -1177.987,E2 -1177.987} C_VEL
LIN {X 0,Y 594.382,Z 748.531,A -85,B 0,C 180,E1 -1178.843,E2 -1178.843} C_VEL
LIN {X 0,Y 594.428,Z 738.085,A -85,B 0,C 180,E1 -1179.7,E2 -1179.7} C_VEL
LIN {X 0,Y 594.485,Z 727.749,A -85,B 0,C 180,E1 -1180.387,E2 -1180.387} C_VEL
LIN {X 0,Y 594.551,Z 716.798,A -85,B 0,C 180,E1 -1180.97,E2 -1180.97} C_VEL
LIN {X 0,Y 594.594,Z 704.72,A -85,B 0,C 180,E1 -1181.464,E2 -1181.464} C_VEL
LIN {X 0,Y 594.629,Z 691.329,A -85,B 0,C 180,E1 -1181.851,E2 -1181.851} C_VEL
LIN {X 0,Y 594.562,Z 679.564,A -85,B 0,C 180,E1 -1182.069,E2 -1182.069} C_VEL
LIN {X 0,Y 594.361,Z 678.031,A -85,B 0,C 180,E1 -1182.116,E2 -1182.116} C_VEL
LIN {X 0,Y 594.396,Z 663.358,A -85,B 0,C 180,E1 -1184.727,E2 -1184.727} C_VEL
LIN {X 0,Y 594.464,Z 647.707,A -85,B 0,C 180,E1 -1187.547,E2 -1187.547} C_VEL
LIN {X 0,Y 594.493,Z 634.012,A -85,B 0,C 180,E1 -1190.05,E2 -1190.05} C_VEL
LIN {X 0,Y 594.619,Z 618.361,A -85,B 0,C 180,E1 -1192.957,E2 -1192.957} C_VEL
LIN {X 0,Y 594.672,Z 604.666,A -85,B 0,C 180,E1 -1195.555,E2 -1195.555} C_VEL
LIN {X 0,Y 594.778,Z 590.971,A -85,B 0,C 180,E1 -1198.207,E2 -1198.207} C_VEL
LIN {X 0,Y 594.886,Z 577.276,A -85,B 0,C 180,E1 -1200.925,E2 -1200.925} C_VEL
LIN {X 0,Y 594.921,Z 566.792,A -85,B 0,C 180,E1 -1202.992,E2 -1202.992} C_VEL
LIN {X 0,Y 594.8,Z 553.491,A -85,B 0,C 180,E1 -1205.586,E2 -1205.586} C_VEL
LIN {X 0,Y 594.356,Z 550.454,A -85,B 0,C 180,E1 -1206.245,E2 -1206.245} C_VEL
LIN {X 0,Y 594.393,Z 550.448,A -85,B 0,C 180,E1 -1208.805,E2 -1208.805} C_VEL
LIN {X 0,Y 594.389,Z 550.448,A -85,B 0,C 180,E1 -1211.849,E2 -1211.849} C_VEL
LIN {X 0,Y 594.368,Z 550.45,A -85,B 0,C 180,E1 -1214.809,E2 -1214.809} C_VEL
LIN {X 0,Y 594.373,Z 550.449,A -85,B 0,C 180,E1 -1217.625,E2 -1217.625} C_VEL
LIN {X 0,Y 594.378,Z 550.451,A -85,B 0,C 180,E1 -1220.319,E2 -1220.319} C_VEL
LIN {X 0,Y 594.39,Z 550.447,A -85,B 0,C 180,E1 -1222.913,E2 -1222.913} C_VEL
LIN {X 0,Y 594.388,Z 550.447,A -85,B 0,C 180,E1 -1225.861,E2 -1225.861} C_VEL
LIN {X 0,Y 594.373,Z 550.45,A -85,B 0,C 180,E1 -1228.65,E2 -1228.65} C_VEL
LIN {X 0,Y 594.388,Z 550.448,A -85,B 0,C 180,E1 -1231.042,E2 -1231.042} C_VEL
LIN {X 0,Y 594.393,Z 550.447,A -85,B 0,C 180,E1 -1233.976,E2 -1233.976} C_VEL
LIN {X 0,Y 594.39,Z 550.447,A -85,B 0,C 180,E1 -1236.296,E2 -1236.296} C_VEL
LIN {X 0,Y 594.409,Z 550.445,A -85,B 0,C 180,E1 -1239.224,E2 -1239.224} C_VEL
LIN {X 0,Y 594.353,Z 550.451,A -85,B 0,C 180,E1 -1242.095,E2 -1242.095} C_VEL
LIN {X 0,Y 594.371,Z 550.449,A -85,B 0,C 180,E1 -1244.219,E2 -1244.219} C_VEL
LIN {X 0,Y 594.383,Z 550.448,A -85,B 0,C 180,E1 -1246.321,E2 -1246.321} C_VEL
LIN {X 0,Y 594.378,Z 550.448,A -85,B 0,C 180,E1 -1249.094,E2 -1249.094} C_VEL
LIN {X 0,Y 594.419,Z 550.446,A -85,B 0,C 180,E1 -1251.843,E2 -1251.843} C_VEL
LIN {X 0,Y 594.393,Z 550.446,A -85,B 0,C 180,E1 -1254.572,E2 -1254.572} C_VEL
LIN {X 0,Y 594.413,Z 550.444,A -85,B 0,C 180,E1 -1257.289,E2 -1257.289} C_VEL
LIN {X 0,Y 594.417,Z 550.446,A -85,B 0,C 180,E1 -1260,E2 -1260} C_VEL
LIN {X 0,Y 594.413,Z 550.444,A -85,B 0,C 180,E1 -1262.71,E2 -1262.71} C_VEL
LIN {X 0,Y 594.392,Z 550.446,A -85,B 0,C 180,E1 -1265.427,E2 -1265.427} C_VEL
LIN {X 0,Y 594.418,Z 550.446,A -85,B 0,C 180,E1 -1268.156,E2 -1268.156} C_VEL
LIN {X 0,Y 594.392,Z 550.446,A -85,B 0,C 180,E1 -1271.073,E2 -1271.073} C_VEL
LIN {X 0,Y 594.386,Z 550.447,A -85,B 0,C 180,E1 -1273.679,E2 -1273.679} C_VEL
LIN {X 0,Y 594.366,Z 550.45,A -85,B 0,C 180,E1 -1275.327,E2 -1275.327} C_VEL
LIN {X 0,Y 593.692,Z 550.534,A -85,B 0,C 180,E1 -1275.893,E2 -1275.893} C_VEL
LIN {X 0,Y 590.823,Z 550.891,A -85,B 0,C 180,E1 -1276.811,E2 -1276.811} C_VEL
LIN {X 0,Y 588.41,Z 551.194,A -85,B 0,C 180,E1 -1277.55,E2 -1277.55} C_VEL
LIN {X 0,Y 587.387,Z 551.319,A -85,B 0,C 180,E1 -1278.12,E2 -1278.12} C_VEL
LIN {X 0,Y 587.311,Z 551.327,A -85,B 0,C 180,E1 -1278.313,E2 -1278.313} C_VEL
LIN {X 0,Y 587.333,Z 551.328,A -85,B 0,C 180,E1 -1281.037,E2 -1281.037} C_VEL
LIN {X 0,Y 587.324,Z 551.329,A -85,B 0,C 180,E1 -1283.258,E2 -1283.258} C_VEL
LIN {X 0,Y 587.338,Z 551.326,A -85,B 0,C 180,E1 -1285.516,E2 -1285.516} C_VEL
LIN {X 0,Y 587.351,Z 551.324,A -85,B 0,C 180,E1 -1287.817,E2 -1287.817} C_VEL
LIN {X 0,Y 587.337,Z 551.327,A -85,B 0,C 180,E1 -1290.509,E2 -1290.509} C_VEL
LIN {X 0,Y 587.336,Z 551.325,A -85,B 0,C 180,E1 -1293.396,E2 -1293.396} C_VEL
LIN {X 0,Y 587.358,Z 551.323,A -85,B 0,C 180,E1 -1295.895,E2 -1295.895} C_VEL
LIN {X 0,Y 587.332,Z 551.328,A -85,B 0,C 180,E1 -1298.479,E2 -1298.479} C_VEL
LIN {X 0,Y 587.338,Z 551.325,A -85,B 0,C 180,E1 -1301.156,E2 -1301.156} C_VEL
LIN {X 0,Y 587.336,Z 551.326,A -85,B 0,C 180,E1 -1304.114,E2 -1304.114} C_VEL
LIN {X 0,Y 587.323,Z 551.327,A -85,B 0,C 180,E1 -1306.994,E2 -1306.994} C_VEL
LIN {X 0,Y 587.323,Z 551.326,A -85,B 0,C 180,E1 -1309.746,E2 -1309.746} C_VEL
LIN {X 0,Y 587.348,Z 551.325,A -85,B 0,C 180,E1 -1312.392,E2 -1312.392} C_VEL
LIN {X 0,Y 587.361,Z 551.322,A -85,B 0,C 180,E1 -1315.78,E2 -1315.78} C_VEL
LIN {X 0,Y 587.356,Z 551.324,A -85,B 0,C 180,E1 -1318.232,E2 -1318.232} C_VEL
LIN {X 0,Y 587.349,Z 551.325,A -85,B 0,C 180,E1 -1320.866,E2 -1320.866} C_VEL
LIN {X 0,Y 587.362,Z 551.322,A -85,B 0,C 180,E1 -1323.818,E2 -1323.818} C_VEL
LIN {X 0,Y 587.34,Z 551.324,A -85,B 0,C 180,E1 -1325.993,E2 -1325.993} C_VEL
LIN {X 0,Y 587.322,Z 551.327,A -85,B 0,C 180,E1 -1328.225,E2 -1328.225} C_VEL
LIN {X 0,Y 587.351,Z 551.326,A -85,B 0,C 180,E1 -1331.151,E2 -1331.151} C_VEL
LIN {X 0,Y 587.33,Z 551.326,A -85,B 0,C 180,E1 -1334.024,E2 -1334.024} C_VEL
LIN {X 0,Y 587.36,Z 551.323,A -85,B 0,C 180,E1 -1336.154,E2 -1336.154} C_VEL
LIN {X 0,Y 587.344,Z 551.324,A -85,B 0,C 180,E1 -1338.962,E2 -1338.962} C_VEL
LIN {X 0,Y 587.365,Z 551.324,A -85,B 0,C 180,E1 -1341.744,E2 -1341.744} C_VEL
LIN {X 0,Y 587.357,Z 551.323,A -85,B 0,C 180,E1 -1344.506,E2 -1344.506} C_VEL
LIN {X 0,Y 587.373,Z 551.321,A -85,B 0,C 180,E1 -1347.256,E2 -1347.256} C_VEL
LIN {X 0,Y 587.384,Z 551.322,A -85,B 0,C 180,E1 -1349.999,E2 -1349.999} C_VEL
LIN {X 0,Y 587.35,Z 551.327,A -85,B 0,C 180,E1 -1352.314,E2 -1352.314} C_VEL
LIN {X 0,Y 587.622,Z 555.871,A -85,B 0,C 180,E1 -1352.484,E2 -1352.484} C_VEL
LIN {X 0,Y 587.538,Z 567.936,A -85,B 0,C 180,E1 -1352.999,E2 -1352.999} C_VEL
LIN {X 0,Y 587.477,Z 578.835,A -85,B 0,C 180,E1 -1353.6,E2 -1353.6} C_VEL
LIN {X 0,Y 587.427,Z 588.853,A -85,B 0,C 180,E1 -1354.288,E2 -1354.288} C_VEL
LIN {X 0,Y 587.361,Z 597.173,A -85,B 0,C 180,E1 -1354.976,E2 -1354.976} C_VEL
LIN {X 0,Y 587.273,Z 605.837,A -85,B 0,C 180,E1 -1355.838,E2 -1355.838} C_VEL
LIN {X 0,Y 587.261,Z 612.565,A -85,B 0,C 180,E1 -1356.641,E2 -1356.641} C_VEL
LIN {X 0,Y 587.228,Z 620.131,A -85,B 0,C 180,E1 -1357.737,E2 -1357.737} C_VEL
LIN {X 0,Y 587.185,Z 626.636,A -85,B 0,C 180,E1 -1358.951,E2 -1358.951} C_VEL
LIN {X 0,Y 587.178,Z 630.925,A -85,B 0,C 180,E1 -1359.994,E2 -1359.994} C_VEL
LIN {X 0,Y 587.159,Z 634.146,A -85,B 0,C 180,E1 -1361.04,E2 -1361.04} C_VEL
LIN {X 0,Y 587.152,Z 635.735,A -85,B 0,C 180,E1 -1361.74,E2 -1361.74} C_VEL
LIN {X 0,Y 587.158,Z 636.887,A -85,B 0,C 180,E1 -1362.441,E2 -1362.441} C_VEL
LIN {X 0,Y 587.143,Z 637.639,A -85,B 0,C 180,E1 -1363.145,E2 -1363.145} C_VEL
LIN {X 0,Y 587.154,Z 637.976,A -85,B 0,C 180,E1 -1364.18,E2 -1364.18} C_VEL
LIN {X 0,Y 587.13,Z 637.352,A -85,B 0,C 180,E1 -1365.268,E2 -1365.268} C_VEL
LIN {X 0,Y 587.156,Z 636.401,A -85,B 0,C 180,E1 -1365.979,E2 -1365.979} C_VEL
LIN {X 0,Y 587.139,Z 634.878,A -85,B 0,C 180,E1 -1366.747,E2 -1366.747} C_VEL
LIN {X 0,Y 587.161,Z 632.023,A -85,B 0,C 180,E1 -1367.771,E2 -1367.771} C_VEL
LIN {X 0,Y 587.176,Z 627.318,A -85,B 0,C 180,E1 -1368.993,E2 -1368.993} C_VEL
LIN {X 0,Y 587.221,Z 620.409,A -85,B 0,C 180,E1 -1370.308,E2 -1370.308} C_VEL
LIN {X 0,Y 587.243,Z 612.885,A -85,B 0,C 180,E1 -1371.408,E2 -1371.408} C_VEL
LIN {X 0,Y 587.304,Z 605.13,A -85,B 0,C 180,E1 -1372.329,E2 -1372.329} C_VEL
LIN {X 0,Y 587.369,Z 595.593,A -85,B 0,C 180,E1 -1373.256,E2 -1373.256} C_VEL
LIN {X 0,Y 587.425,Z 584.995,A -85,B 0,C 180,E1 -1374.087,E2 -1374.087} C_VEL
LIN {X 0,Y 587.512,Z 574.415,A -85,B 0,C 180,E1 -1374.75,E2 -1374.75} C_VEL
LIN {X 0,Y 587.574,Z 563.065,A -85,B 0,C 180,E1 -1375.315,E2 -1375.315} C_VEL
LIN {X 0,Y 587.64,Z 553.348,A -85,B 0,C 180,E1 -1375.691,E2 -1375.691} C_VEL
LIN {X 0,Y 587.341,Z 551.328,A -85,B 0,C 180,E1 -1375.777,E2 -1375.777} C_VEL
LIN {X 0,Y 587.322,Z 551.327,A -85,B 0,C 180,E1 -1378.596,E2 -1378.596} C_VEL
LIN {X 0,Y 587.341,Z 551.324,A -85,B 0,C 180,E1 -1380.965,E2 -1380.965} C_VEL
LIN {X 0,Y 587.332,Z 551.325,A -85,B 0,C 180,E1 -1383.396,E2 -1383.396} C_VEL
LIN {X 0,Y 587.313,Z 551.328,A -85,B 0,C 180,E1 -1385.897,E2 -1385.897} C_VEL
LIN {X 0,Y 587.33,Z 551.328,A -85,B 0,C 180,E1 -1388.478,E2 -1388.478} C_VEL
LIN {X 0,Y 587.35,Z 551.325,A -85,B 0,C 180,E1 -1391.554,E2 -1391.554} C_VEL
LIN {X 0,Y 587.448,Z 558.889,A -85,B 0,C 180,E1 -1394.126,E2 -1394.126} C_VEL
LIN {X 0,Y 587.455,Z 567.415,A -85,B 0,C 180,E1 -1397.007,E2 -1397.007} C_VEL
LIN {X 0,Y 587.39,Z 575.279,A -85,B 0,C 180,E1 -1399.752,E2 -1399.752} C_VEL
LIN {X 0,Y 587.351,Z 583.024,A -85,B 0,C 180,E1 -1402.393,E2 -1402.393} C_VEL
LIN {X 0,Y 587.338,Z 590.663,A -85,B 0,C 180,E1 -1404.945,E2 -1404.945} C_VEL
LIN {X 0,Y 587.295,Z 598.201,A -85,B 0,C 180,E1 -1407.419,E2 -1407.419} C_VEL
LIN {X 0,Y 587.252,Z 606.882,A -85,B 0,C 180,E1 -1410.221,E2 -1410.221} C_VEL
LIN {X 0,Y 587.198,Z 615.45,A -85,B 0,C 180,E1 -1412.948,E2 -1412.948} C_VEL
LIN {X 0,Y 587.209,Z 621.472,A -85,B 0,C 180,E1 -1414.845,E2 -1414.845} C_VEL
LIN {X 0,Y 587.731,Z 626.665,A -85,B 0,C 180,E1 -1414.952,E2 -1414.952} C_VEL
LIN {X 0,Y 587.647,Z 640.528,A -85,B 0,C 180,E1 -1415.303,E2 -1415.303} C_VEL
LIN {X 0,Y 587.599,Z 652.284,A -85,B 0,C 180,E1 -1415.742,E2 -1415.742} C_VEL
LIN {X 0,Y 587.49,Z 663.352,A -85,B 0,C 180,E1 -1416.282,E2 -1416.282} C_VEL
LIN {X 0,Y 587.449,Z 674.744,A -85,B 0,C 180,E1 -1416.987,E2 -1416.987} C_VEL
LIN {X 0,Y 587.397,Z 684.846,A -85,B 0,C 180,E1 -1417.767,E2 -1417.767} C_VEL
LIN {X 0,Y 587.309,Z 693.587,A -85,B 0,C 180,E1 -1418.594,E2 -1418.594} C_VEL
LIN {X 0,Y 587.252,Z 701.561,A -85,B 0,C 180,E1 -1419.51,E2 -1419.51} C_VEL
LIN {X 0,Y 587.227,Z 709.151,A -85,B 0,C 180,E1 -1420.582,E2 -1420.582} C_VEL
LIN {X 0,Y 587.217,Z 714.451,A -85,B 0,C 180,E1 -1421.509,E2 -1421.509} C_VEL
LIN {X 0,Y 587.167,Z 719.379,A -85,B 0,C 180,E1 -1422.589,E2 -1422.589} C_VEL
LIN {X 0,Y 587.156,Z 723.098,A -85,B 0,C 180,E1 -1423.663,E2 -1423.663} C_VEL
LIN {X 0,Y 587.142,Z 725.719,A -85,B 0,C 180,E1 -1424.732,E2 -1424.732} C_VEL
LIN {X 0,Y 587.148,Z 727.348,A -85,B 0,C 180,E1 -1425.819,E2 -1425.819} C_VEL
LIN {X 0,Y 587.14,Z 727.963,A -85,B 0,C 180,E1 -1426.855,E2 -1426.855} C_VEL
LIN {X 0,Y 587.156,Z 727.868,A -85,B 0,C 180,E1 -1427.558,E2 -1427.558} C_VEL
LIN {X 0,Y 587.149,Z 727.361,A -85,B 0,C 180,E1 -1428.259,E2 -1428.259} C_VEL
LIN {X 0,Y 587.191,Z 726.434,A -85,B 0,C 180,E1 -1428.96,E2 -1428.96} C_VEL
LIN {X 0,Y 587.14,Z 725.089,A -85,B 0,C 180,E1 -1429.657,E2 -1429.657} C_VEL
LIN {X 0,Y 587.185,Z 722.249,A -85,B 0,C 180,E1 -1430.702,E2 -1430.702} C_VEL
LIN {X 0,Y 587.185,Z 718.383,A -85,B 0,C 180,E1 -1431.742,E2 -1431.742} C_VEL
LIN {X 0,Y 587.209,Z 713.4,A -85,B 0,C 180,E1 -1432.781,E2 -1432.781} C_VEL
LIN {X 0,Y 587.23,Z 707.154,A -85,B 0,C 180,E1 -1433.817,E2 -1433.817} C_VEL
LIN {X 0,Y 587.302,Z 699.371,A -85,B 0,C 180,E1 -1434.851,E2 -1434.851} C_VEL
LIN {X 0,Y 587.328,Z 689.688,A -85,B 0,C 180,E1 -1435.883,E2 -1435.883} C_VEL
LIN {X 0,Y 587.412,Z 679.675,A -85,B 0,C 180,E1 -1436.742,E2 -1436.742} C_VEL
LIN {X 0,Y 587.473,Z 668.446,A -85,B 0,C 180,E1 -1437.515,E2 -1437.515} C_VEL
LIN {X 0,Y 587.553,Z 657.453,A -85,B 0,C 180,E1 -1438.115,E2 -1438.115} C_VEL
LIN {X 0,Y 587.638,Z 646.362,A -85,B 0,C 180,E1 -1438.587,E2 -1438.587} C_VEL
LIN {X 0,Y 587.699,Z 633.965,A -85,B 0,C 180,E1 -1438.972,E2 -1438.972} C_VEL
LIN {X 0,Y 587.463,Z 623.091,A -85,B 0,C 180,E1 -1439.208,E2 -1439.208} C_VEL
LIN {X 0,Y 587.217,Z 621.405,A -85,B 0,C 180,E1 -1439.272,E2 -1439.272} C_VEL
LIN {X 0,Y 587.284,Z 613.687,A -85,B 0,C 180,E1 -1441.715,E2 -1441.715} C_VEL
LIN {X 0,Y 587.274,Z 604.053,A -85,B 0,C 180,E1 -1444.806,E2 -1444.806} C_VEL
LIN {X 0,Y 587.295,Z 595.59,A -85,B 0,C 180,E1 -1447.564,E2 -1447.564} C_VEL
LIN {X 0,Y 587.336,Z 587.224,A -85,B 0,C 180,E1 -1450.34,E2 -1450.34} C_VEL
LIN {X 0,Y 587.393,Z 578.957,A -85,B 0,C 180,E1 -1453.14,E2 -1453.14} C_VEL
LIN {X 0,Y 587.423,Z 570.795,A -85,B 0,C 180,E1 -1455.973,E2 -1455.973} C_VEL
LIN {X 0,Y 587.434,Z 564.433,A -85,B 0,C 180,E1 -1458.123,E2 -1458.123} C_VEL
LIN {X 0,Y 587.281,Z 554.833,A -85,B 0,C 180,E1 -1461.04,E2 -1461.04} C_VEL
LIN {X 0,Y 587.283,Z 551.334,A -85,B 0,C 180,E1 -1462.053,E2 -1462.053} C_VEL
LIN {X 0,Y 587.347,Z 551.326,A -85,B 0,C 180,E1 -1464.759,E2 -1464.759} C_VEL
LIN {X 0,Y 587.335,Z 551.329,A -85,B 0,C 180,E1 -1467.046,E2 -1467.046} C_VEL
LIN {X 0,Y 587.348,Z 551.325,A -85,B 0,C 180,E1 -1469.38,E2 -1469.38} C_VEL
LIN {X 0,Y 587.355,Z 551.324,A -85,B 0,C 180,E1 -1471.839,E2 -1471.839} C_VEL
LIN {X 0,Y 587.354,Z 551.326,A -85,B 0,C 180,E1 -1474.35,E2 -1474.35} C_VEL
LIN {X 0,Y 587.349,Z 551.324,A -85,B 0,C 180,E1 -1476.747,E2 -1476.747} C_VEL
LIN {X 0,Y 587.344,Z 551.327,A -85,B 0,C 180,E1 -1479.36,E2 -1479.36} C_VEL
LIN {X 0,Y 587.33,Z 551.326,A -85,B 0,C 180,E1 -1482.109,E2 -1482.109} C_VEL
LIN {X 0,Y 587.312,Z 551.329,A -85,B 0,C 180,E1 -1485.09,E2 -1485.09} C_VEL
LIN {X 0,Y 587.35,Z 551.325,A -85,B 0,C 180,E1 -1487.928,E2 -1487.928} C_VEL
LIN {X 0,Y 587.334,Z 551.328,A -85,B 0,C 180,E1 -1491.059,E2 -1491.059} C_VEL
LIN {X 0,Y 587.383,Z 551.466,A -85,B 0,C 180,E1 -1493.736,E2 -1493.736} C_VEL
LIN {X 0,Y 587.927,Z 556.105,A -85,B 0,C 180,E1 -1494.69,E2 -1494.69} C_VEL
LIN {X 0,Y 587.996,Z 570.318,A -85,B 0,C 180,E1 -1497.463,E2 -1497.463} C_VEL
LIN {X 0,Y 588.002,Z 580.332,A -85,B 0,C 180,E1 -1499.381,E2 -1499.381} C_VEL
LIN {X 0,Y 587.849,Z 594.565,A -85,B 0,C 180,E1 -1502.215,E2 -1502.215} C_VEL
LIN {X 0,Y 587.716,Z 608.282,A -85,B 0,C 180,E1 -1504.881,E2 -1504.881} C_VEL
LIN {X 0,Y 587.611,Z 622.032,A -85,B 0,C 180,E1 -1507.498,E2 -1507.498} C_VEL
LIN {X 0,Y 587.522,Z 635.782,A -85,B 0,C 180,E1 -1510.068,E2 -1510.068} C_VEL
LIN {X 0,Y 587.412,Z 651.38,A -85,B 0,C 180,E1 -1512.935,E2 -1512.935} C_VEL
LIN {X 0,Y 587.333,Z 666.945,A -85,B 0,C 180,E1 -1515.753,E2 -1515.753} C_VEL
LIN {X 0,Y 587.315,Z 678.139,A -85,B 0,C 180,E1 -1517.76,E2 -1517.76} C_VEL
LIN {X 0,Y 587.743,Z 683.985,A -85,B 0,C 180,E1 -1517.856,E2 -1517.856} C_VEL
LIN {X 0,Y 587.665,Z 697.244,A -85,B 0,C 180,E1 -1518.161,E2 -1518.161} C_VEL
LIN {X 0,Y 587.623,Z 709.893,A -85,B 0,C 180,E1 -1518.595,E2 -1518.595} C_VEL
LIN {X 0,Y 587.537,Z 721.646,A -85,B 0,C 180,E1 -1519.141,E2 -1519.141} C_VEL
LIN {X 0,Y 587.449,Z 733.211,A -85,B 0,C 180,E1 -1519.837,E2 -1519.837} C_VEL
LIN {X 0,Y 587.366,Z 743.605,A -85,B 0,C 180,E1 -1520.618,E2 -1520.618} C_VEL
LIN {X 0,Y 587.321,Z 752.119,A -85,B 0,C 180,E1 -1521.398,E2 -1521.398} C_VEL
LIN {X 0,Y 587.273,Z 759.966,A -85,B 0,C 180,E1 -1522.263,E2 -1522.263} C_VEL
LIN {X 0,Y 587.23,Z 766.475,A -85,B 0,C 180,E1 -1523.127,E2 -1523.127} C_VEL
LIN {X 0,Y 587.236,Z 772.87,A -85,B 0,C 180,E1 -1524.162,E2 -1524.162} C_VEL
LIN {X 0,Y 587.147,Z 777.953,A -85,B 0,C 180,E1 -1525.194,E2 -1525.194} C_VEL
LIN {X 0,Y 587.212,Z 781.898,A -85,B 0,C 180,E1 -1526.226,E2 -1526.226} C_VEL
LIN {X 0,Y 587.132,Z 784.81,A -85,B 0,C 180,E1 -1527.256,E2 -1527.256} C_VEL
LIN {X 0,Y 587.138,Z 786.202,A -85,B 0,C 180,E1 -1527.943,E2 -1527.943} C_VEL
LIN {X 0,Y 587.14,Z 787.785,A -85,B 0,C 180,E1 -1529.315,E2 -1529.315} C_VEL
LIN {X 0,Y 587.137,Z 788,A -85,B 0,C 180,E1 -1530.001,E2 -1530.001} C_VEL
LIN {X 0,Y 587.147,Z 787.184,A -85,B 0,C 180,E1 -1531.372,E2 -1531.372} C_VEL
LIN {X 0,Y 587.138,Z 786.201,A -85,B 0,C 180,E1 -1532.059,E2 -1532.059} C_VEL
LIN {X 0,Y 587.132,Z 784.808,A -85,B 0,C 180,E1 -1532.745,E2 -1532.745} C_VEL
LIN {X 0,Y 587.212,Z 781.894,A -85,B 0,C 180,E1 -1533.775,E2 -1533.775} C_VEL
LIN {X 0,Y 587.147,Z 777.947,A -85,B 0,C 180,E1 -1534.807,E2 -1534.807} C_VEL
LIN {X 0,Y 587.217,Z 771.874,A -85,B 0,C 180,E1 -1536.012,E2 -1536.012} C_VEL
LIN {X 0,Y 587.246,Z 765.232,A -85,B 0,C 180,E1 -1537.047,E2 -1537.047} C_VEL
LIN {X 0,Y 587.3,Z 756.985,A -85,B 0,C 180,E1 -1538.084,E2 -1538.084} C_VEL
LIN {X 0,Y 587.344,Z 748.531,A -85,B 0,C 180,E1 -1538.95,E2 -1538.95} C_VEL
LIN {X 0,Y 587.414,Z 738.086,A -85,B 0,C 180,E1 -1539.817,E2 -1539.817} C_VEL
LIN {X 0,Y 587.5,Z 727.75,A -85,B 0,C 180,E1 -1540.512,E2 -1540.512} C_VEL
LIN {X 0,Y 587.565,Z 716.019,A -85,B 0,C 180,E1 -1541.139,E2 -1541.139} C_VEL
LIN {X 0,Y 587.624,Z 703.608,A -85,B 0,C 180,E1 -1541.639,E2 -1541.639} C_VEL
LIN {X 0,Y 587.712,Z 690.414,A -85,B 0,C 180,E1 -1542.014,E2 -1542.014} C_VEL
LIN {X 0,Y 587.504,Z 679.564,A -85,B 0,C 180,E1 -1542.216,E2 -1542.216} C_VEL
LIN {X 0,Y 587.32,Z 678.031,A -85,B 0,C 180,E1 -1542.264,E2 -1542.264} C_VEL
LIN {X 0,Y 587.383,Z 661.402,A -85,B 0,C 180,E1 -1545.262,E2 -1545.262} C_VEL
LIN {X 0,Y 587.464,Z 645.751,A -85,B 0,C 180,E1 -1548.123,E2 -1548.123} C_VEL
LIN {X 0,Y 587.557,Z 630.099,A -85,B 0,C 180,E1 -1551.03,E2 -1551.03} C_VEL
LIN {X 0,Y 587.644,Z 616.404,A -85,B 0,C 180,E1 -1553.619,E2 -1553.619} C_VEL
LIN {X 0,Y 587.792,Z 602.665,A -85,B 0,C 180,E1 -1556.266,E2 -1556.266} C_VEL
LIN {X 0,Y 587.933,Z 587.623,A -85,B 0,C 180,E1 -1559.235,E2 -1559.235} C_VEL
LIN {X 0,Y 587.996,Z 575.068,A -85,B 0,C 180,E1 -1561.73,E2 -1561.73} C_VEL
LIN {X 0,Y 587.92,Z 561.052,A -85,B 0,C 180,E1 -1564.429,E2 -1564.429} C_VEL
LIN {X 0,Y 587.872,Z 554.014,A -85,B 0,C 180,E1 -1565.86,E2 -1565.86} C_VEL
LIN {X 0,Y 587.348,Z 551.327,A -85,B 0,C 180,E1 -1566.481,E2 -1566.481} C_VEL
LIN {X 0,Y 587.352,Z 551.324,A -85,B 0,C 180,E1 -1569.359,E2 -1569.359} C_VEL
LIN {X 0,Y 587.34,Z 551.328,A -85,B 0,C 180,E1 -1572.108,E2 -1572.108} C_VEL
LIN {X 0,Y 587.321,Z 551.327,A -85,B 0,C 180,E1 -1575.089,E2 -1575.089} C_VEL
LIN {X 0,Y 587.358,Z 551.326,A -85,B 0,C 180,E1 -1577.928,E2 -1577.928} C_VEL
LIN {X 0,Y 587.321,Z 551.327,A -85,B 0,C 180,E1 -1581.06,E2 -1581.06} C_VEL
LIN {X 0,Y 587.359,Z 551.322,A -85,B 0,C 180,E1 -1583.292,E2 -1583.292} C_VEL
LIN {X 0,Y 587.371,Z 551.321,A -85,B 0,C 180,E1 -1585.78,E2 -1585.78} C_VEL
LIN {X 0,Y 587.343,Z 551.325,A -85,B 0,C 180,E1 -1588.231,E2 -1588.231} C_VEL
LIN {X 0,Y 587.354,Z 551.325,A -85,B 0,C 180,E1 -1590.866,E2 -1590.866} C_VEL
LIN {X 0,Y 587.365,Z 551.321,A -85,B 0,C 180,E1 -1593.818,E2 -1593.818} C_VEL
LIN {X 0,Y 587.338,Z 551.325,A -85,B 0,C 180,E1 -1595.993,E2 -1595.993} C_VEL
LIN {X 0,Y 587.327,Z 551.326,A -85,B 0,C 180,E1 -1598.226,E2 -1598.226} C_VEL
LIN {X 0,Y 587.353,Z 551.325,A -85,B 0,C 180,E1 -1601.151,E2 -1601.151} C_VEL
LIN {X 0,Y 587.329,Z 551.326,A -85,B 0,C 180,E1 -1604.025,E2 -1604.025} C_VEL
LIN {X 0,Y 587.362,Z 551.324,A -85,B 0,C 180,E1 -1606.154,E2 -1606.154} C_VEL
LIN {X 0,Y 587.344,Z 551.324,A -85,B 0,C 180,E1 -1608.962,E2 -1608.962} C_VEL
LIN {X 0,Y 587.373,Z 551.323,A -85,B 0,C 180,E1 -1611.745,E2 -1611.745} C_VEL
LIN {X 0,Y 587.359,Z 551.323,A -85,B 0,C 180,E1 -1614.507,E2 -1614.507} C_VEL
LIN {X 0,Y 587.378,Z 551.32,A -85,B 0,C 180,E1 -1617.256,E2 -1617.256} C_VEL
LIN {X 0,Y 587.386,Z 551.322,A -85,B 0,C 180,E1 -1620,E2 -1620} C_VEL
LIN {X 0,Y 587.378,Z 551.32,A -85,B 0,C 180,E1 -1622.743,E2 -1622.743} C_VEL
LIN {X 0,Y 587.358,Z 551.323,A -85,B 0,C 180,E1 -1625.493,E2 -1625.493} C_VEL
LIN {X 0,Y 587.37,Z 551.324,A -85,B 0,C 180,E1 -1628.255,E2 -1628.255} C_VEL
LIN {X 0,Y 587.351,Z 551.323,A -85,B 0,C 180,E1 -1631.133,E2 -1631.133} C_VEL
LIN {X 0,Y 587.368,Z 551.322,A -85,B 0,C 180,E1 -1634.26,E2 -1634.26} C_VEL
LIN {X 0,Y 587.35,Z 551.326,A -85,B 0,C 180,E1 -1637.406,E2 -1637.406} C_VEL
LIN {X 0,Y 587.311,Z 551.327,A -85,B 0,C 180,E1 -1638.313,E2 -1638.313} C_VEL
LIN {X 0,Y 586.67,Z 551.41,A -85,B 0,C 180,E1 -1638.885,E2 -1638.885} C_VEL
LIN {X 0,Y 583.845,Z 551.763,A -85,B 0,C 180,E1 -1639.813,E2 -1639.813} C_VEL
LIN {X 0,Y 581.433,Z 552.063,A -85,B 0,C 180,E1 -1640.56,E2 -1640.56} C_VEL
LIN {X 0,Y 580.38,Z 552.193,A -85,B 0,C 180,E1 -1641.137,E2 -1641.137} C_VEL
LIN {X 0,Y 580.286,Z 552.204,A -85,B 0,C 180,E1 -1641.332,E2 -1641.332} C_VEL
LIN {X 0,Y 580.281,Z 552.205,A -85,B 0,C 180,E1 -1643.558,E2 -1643.558} C_VEL
LIN {X 0,Y 580.296,Z 552.204,A -85,B 0,C 180,E1 -1645.848,E2 -1645.848} C_VEL
LIN {X 0,Y 580.303,Z 552.203,A -85,B 0,C 180,E1 -1648.185,E2 -1648.185} C_VEL
LIN {X 0,Y 580.285,Z 552.204,A -85,B 0,C 180,E1 -1650.694,E2 -1650.694} C_VEL
LIN {X 0,Y 580.305,Z 552.2,A -85,B 0,C 180,E1 -1653.316,E2 -1653.316} C_VEL
LIN {X 0,Y 580.328,Z 552.198,A -85,B 0,C 180,E1 -1655.767,E2 -1655.767} C_VEL
LIN {X 0,Y 580.29,Z 552.203,A -85,B 0,C 180,E1 -1658.146,E2 -1658.146} C_VEL
LIN {X 0,Y 580.3,Z 552.205,A -85,B 0,C 180,E1 -1660.843,E2 -1660.843} C_VEL
LIN {X 0,Y 580.289,Z 552.203,A -85,B 0,C 180,E1 -1663.656,E2 -1663.656} C_VEL
LIN {X 0,Y 580.286,Z 552.206,A -85,B 0,C 180,E1 -1666.608,E2 -1666.608} C_VEL
LIN {X 0,Y 580.303,Z 552.203,A -85,B 0,C 180,E1 -1669.157,E2 -1669.157} C_VEL
LIN {X 0,Y 580.292,Z 552.202,A -85,B 0,C 180,E1 -1671.926,E2 -1671.926} C_VEL
LIN {X 0,Y 580.251,Z 552.208,A -85,B 0,C 180,E1 -1674.452,E2 -1674.452} C_VEL
LIN {X 0,Y 580.293,Z 552.204,A -85,B 0,C 180,E1 -1676.975,E2 -1676.975} C_VEL
LIN {X 0,Y 580.304,Z 552.203,A -85,B 0,C 180,E1 -1679.425,E2 -1679.425} C_VEL
LIN {X 0,Y 580.299,Z 552.203,A -85,B 0,C 180,E1 -1682.141,E2 -1682.141} C_VEL
LIN {X 0,Y 580.323,Z 552.201,A -85,B 0,C 180,E1 -1685.269,E2 -1685.269} C_VEL
LIN {X 0,Y 580.274,Z 552.206,A -85,B 0,C 180,E1 -1687.947,E2 -1687.947} C_VEL
LIN {X 0,Y 580.32,Z 552.2,A -85,B 0,C 180,E1 -1690.914,E2 -1690.914} C_VEL
LIN {X 0,Y 580.282,Z 552.205,A -85,B 0,C 180,E1 -1693.825,E2 -1693.825} C_VEL
LIN {X 0,Y 580.327,Z 552.201,A -85,B 0,C 180,E1 -1695.983,E2 -1695.983} C_VEL
LIN {X 0,Y 580.305,Z 552.201,A -85,B 0,C 180,E1 -1698.826,E2 -1698.826} C_VEL
LIN {X 0,Y 580.328,Z 552.2,A -85,B 0,C 180,E1 -1701.643,E2 -1701.643} C_VEL
LIN {X 0,Y 580.324,Z 552.199,A -85,B 0,C 180,E1 -1704.44,E2 -1704.44} C_VEL
LIN {X 0,Y 580.34,Z 552.197,A -85,B 0,C 180,E1 -1707.223,E2 -1707.223} C_VEL
LIN {X 0,Y 580.353,Z 552.198,A -85,B 0,C 180,E1 -1709.999,E2 -1709.999} C_VEL
LIN {X 0,Y 580.311,Z 552.203,A -85,B 0,C 180,E1 -1712.212,E2 -1712.212} C_VEL
LIN {X 0,Y 580.655,Z 555.784,A -85,B 0,C 180,E1 -1712.34,E2 -1712.34} C_VEL
LIN {X 0,Y 580.584,Z 567.865,A -85,B 0,C 180,E1 -1712.861,E2 -1712.861} C_VEL
LIN {X 0,Y 580.48,Z 578.785,A -85,B 0,C 180,E1 -1713.47,E2 -1713.47} C_VEL
LIN {X 0,Y 580.392,Z 588.806,A -85,B 0,C 180,E1 -1714.166,E2 -1714.166} C_VEL
LIN {X 0,Y 580.331,Z 597.128,A -85,B 0,C 180,E1 -1714.862,E2 -1714.862} C_VEL
LIN {X 0,Y 580.213,Z 605.802,A -85,B 0,C 180,E1 -1715.734,E2 -1715.734} C_VEL
LIN {X 0,Y 580.19,Z 613.275,A -85,B 0,C 180,E1 -1716.645,E2 -1716.645} C_VEL
LIN {X 0,Y 580.143,Z 620.105,A -85,B 0,C 180,E1 -1717.657,E2 -1717.657} C_VEL
LIN {X 0,Y 580.109,Z 625.808,A -85,B 0,C 180,E1 -1718.709,E2 -1718.709} C_VEL
LIN {X 0,Y 580.081,Z 630.291,A -85,B 0,C 180,E1 -1719.765,E2 -1719.765} C_VEL
LIN {X 0,Y 580.071,Z 634.334,A -85,B 0,C 180,E1 -1721.077,E2 -1721.077} C_VEL
LIN {X 0,Y 580.051,Z 636.081,A -85,B 0,C 180,E1 -1721.886,E2 -1721.886} C_VEL
LIN {X 0,Y 580.058,Z 637.753,A -85,B 0,C 180,E1 -1723.308,E2 -1723.308} C_VEL
LIN {X 0,Y 580.045,Z 637.964,A -85,B 0,C 180,E1 -1724.234,E2 -1724.234} C_VEL
LIN {X 0,Y 580.029,Z 637.152,A -85,B 0,C 180,E1 -1725.459,E2 -1725.459} C_VEL
LIN {X 0,Y 580.063,Z 636.121,A -85,B 0,C 180,E1 -1726.18,E2 -1726.18} C_VEL
LIN {X 0,Y 580.062,Z 634.592,A -85,B 0,C 180,E1 -1726.904,E2 -1726.904} C_VEL
LIN {X 0,Y 580.079,Z 631.449,A -85,B 0,C 180,E1 -1727.995,E2 -1727.995} C_VEL
LIN {X 0,Y 580.092,Z 627.143,A -85,B 0,C 180,E1 -1729.093,E2 -1729.093} C_VEL
LIN {X 0,Y 580.129,Z 620.423,A -85,B 0,C 180,E1 -1730.382,E2 -1730.382} C_VEL
LIN {X 0,Y 580.187,Z 612.898,A -85,B 0,C 180,E1 -1731.495,E2 -1731.495} C_VEL
LIN {X 0,Y 580.251,Z 605.144,A -85,B 0,C 180,E1 -1732.427,E2 -1732.427} C_VEL
LIN {X 0,Y 580.325,Z 597.302,A -85,B 0,C 180,E1 -1733.212,E2 -1733.212} C_VEL
LIN {X 0,Y 580.4,Z 587.487,A -85,B 0,C 180,E1 -1734.026,E2 -1734.026} C_VEL
LIN {X 0,Y 580.513,Z 576.339,A -85,B 0,C 180,E1 -1734.772,E2 -1734.772} C_VEL
LIN {X 0,Y 580.601,Z 564.212,A -85,B 0,C 180,E1 -1735.401,E2 -1735.401} C_VEL
LIN {X 0,Y 580.53,Z 553.323,A -85,B 0,C 180,E1 -1735.837,E2 -1735.837} C_VEL
LIN {X 0,Y 580.328,Z 552.201,A -85,B 0,C 180,E1 -1735.884,E2 -1735.884} C_VEL
LIN {X 0,Y 580.296,Z 552.205,A -85,B 0,C 180,E1 -1738.185,E2 -1738.185} C_VEL
LIN {X 0,Y 580.296,Z 552.203,A -85,B 0,C 180,E1 -1740.697,E2 -1740.697} C_VEL
LIN {X 0,Y 580.3,Z 552.201,A -85,B 0,C 180,E1 -1743.316,E2 -1743.316} C_VEL
LIN {X 0,Y 580.27,Z 552.205,A -85,B 0,C 180,E1 -1745.76,E2 -1745.76} C_VEL
LIN {X 0,Y 580.285,Z 552.203,A -85,B 0,C 180,E1 -1748.145,E2 -1748.145} C_VEL
LIN {X 0,Y 580.315,Z 552.202,A -85,B 0,C 180,E1 -1750.841,E2 -1750.841} C_VEL
LIN {X 0,Y 580.304,Z 552.334,A -85,B 0,C 180,E1 -1751.582,E2 -1751.582} C_VEL
LIN {X 0,Y 580.424,Z 559.673,A -85,B 0,C 180,E1 -1754.025,E2 -1754.025} C_VEL
LIN {X 0,Y 580.416,Z 568.128,A -85,B 0,C 180,E1 -1756.95,E2 -1756.95} C_VEL
LIN {X 0,Y 580.409,Z 574.624,A -85,B 0,C 180,E1 -1759.166,E2 -1759.166} C_VEL
LIN {X 0,Y 580.331,Z 582.574,A -85,B 0,C 180,E1 -1761.92,E2 -1761.92} C_VEL
LIN {X 0,Y 580.292,Z 590.047,A -85,B 0,C 180,E1 -1764.456,E2 -1764.456} C_VEL
LIN {X 0,Y 580.235,Z 598.853,A -85,B 0,C 180,E1 -1767.385,E2 -1767.385} C_VEL
LIN {X 0,Y 580.186,Z 607.534,A -85,B 0,C 180,E1 -1770.222,E2 -1770.222} C_VEL
LIN {X 0,Y 580.133,Z 616.101,A -85,B 0,C 180,E1 -1772.981,E2 -1772.981} C_VEL
LIN {X 0,Y 580.147,Z 621.482,A -85,B 0,C 180,E1 -1774.697,E2 -1774.697} C_VEL
LIN {X 0,Y 580.796,Z 627.604,A -85,B 0,C 180,E1 -1774.824,E2 -1774.824} C_VEL
LIN {X 0,Y 580.698,Z 640.439,A -85,B 0,C 180,E1 -1775.158,E2 -1775.158} C_VEL
LIN {X 0,Y 580.615,Z 652.779,A -85,B 0,C 180,E1 -1775.627,E2 -1775.627} C_VEL
LIN {X 0,Y 580.49,Z 663.651,A -85,B 0,C 180,E1 -1776.167,E2 -1776.167} C_VEL
LIN {X 0,Y 580.427,Z 674.513,A -85,B 0,C 180,E1 -1776.849,E2 -1776.849} C_VEL
LIN {X 0,Y 580.364,Z 685.04,A -85,B 0,C 180,E1 -1777.67,E2 -1777.67} C_VEL
LIN {X 0,Y 580.254,Z 693.743,A -85,B 0,C 180,E1 -1778.507,E2 -1778.507} C_VEL
LIN {X 0,Y 580.183,Z 701.691,A -85,B 0,C 180,E1 -1779.434,E2 -1779.434} C_VEL
LIN {X 0,Y 580.171,Z 708.343,A -85,B 0,C 180,E1 -1780.376,E2 -1780.376} C_VEL
LIN {X 0,Y 580.145,Z 713.585,A -85,B 0,C 180,E1 -1781.275,E2 -1781.275} C_VEL
LIN {X 0,Y 580.089,Z 718.702,A -85,B 0,C 180,E1 -1782.369,E2 -1782.369} C_VEL
LIN {X 0,Y 580.05,Z 721.7,A -85,B 0,C 180,E1 -1783.168,E2 -1783.168} C_VEL
LIN {X 0,Y 580.071,Z 723.678,A -85,B 0,C 180,E1 -1783.82,E2 -1783.82} C_VEL
LIN {X 0,Y 580.06,Z 725.382,A -85,B 0,C 180,E1 -1784.541,E2 -1784.541} C_VEL
LIN {X 0,Y 580.056,Z 727.296,A -85,B 0,C 180,E1 -1785.758,E2 -1785.758} C_VEL
LIN {X 0,Y 580.054,Z 727.927,A -85,B 0,C 180,E1 -1786.691,E2 -1786.691} C_VEL
LIN {X 0,Y 580.046,Z 727.926,A -85,B 0,C 180,E1 -1787.403,E2 -1787.403} C_VEL
LIN {X 0,Y 580.047,Z 727.531,A -85,B 0,C 180,E1 -1788.114,E2 -1788.114} C_VEL
LIN {X 0,Y 580.101,Z 726.56,A -85,B 0,C 180,E1 -1788.904,E2 -1788.904} C_VEL
LIN {X 0,Y 580.06,Z 723.77,A -85,B 0,C 180,E1 -1790.234,E2 -1790.234} C_VEL
LIN {X 0,Y 580.084,Z 720.415,A -85,B 0,C 180,E1 -1791.29,E2 -1791.29} C_VEL
LIN {X 0,Y 580.111,Z 715.986,A -85,B 0,C 180,E1 -1792.342,E2 -1792.342} C_VEL
LIN {X 0,Y 580.142,Z 710.378,A -85,B 0,C 180,E1 -1793.389,E2 -1793.389} C_VEL
LIN {X 0,Y 580.159,Z 703.339,A -85,B 0,C 180,E1 -1794.439,E2 -1794.439} C_VEL
LIN {X 0,Y 580.266,Z 694.646,A -85,B 0,C 180,E1 -1795.485,E2 -1795.485} C_VEL
LIN {X 0,Y 580.339,Z 684.79,A -85,B 0,C 180,E1 -1796.442,E2 -1796.442} C_VEL
LIN {X 0,Y 580.433,Z 674.76,A -85,B 0,C 180,E1 -1797.224,E2 -1797.224} C_VEL
LIN {X 0,Y 580.512,Z 663.711,A -85,B 0,C 180,E1 -1797.919,E2 -1797.919} C_VEL
LIN {X 0,Y 580.594,Z 653.303,A -85,B 0,C 180,E1 -1798.44,E2 -1798.44} C_VEL
LIN {X 0,Y 580.687,Z 642.159,A -85,B 0,C 180,E1 -1798.873,E2 -1798.873} C_VEL
LIN {X 0,Y 580.782,Z 628.845,A -85,B 0,C 180,E1 -1799.242,E2 -1799.242} C_VEL
LIN {X 0,Y 580.438,Z 623.484,A -85,B 0,C 180,E1 -1799.35,E2 -1799.35} C_VEL
LIN {X 0,Y 580.153,Z 621.499,A -85,B 0,C 180,E1 -1799.393,E2 -1799.393} C_VEL
LIN {X 0,Y 580.139,Z 613.118,A -85,B 0,C 180,E1 -1802.083,E2 -1802.083} C_VEL
LIN {X 0,Y 580.22,Z 604.556,A -85,B 0,C 180,E1 -1804.864,E2 -1804.864} C_VEL
LIN {X 0,Y 580.237,Z 596.096,A -85,B 0,C 180,E1 -1807.657,E2 -1807.657} C_VEL
LIN {X 0,Y 580.309,Z 587.731,A -85,B 0,C 180,E1 -1810.467,E2 -1810.467} C_VEL
LIN {X 0,Y 580.356,Z 579.47,A -85,B 0,C 180,E1 -1813.302,E2 -1813.302} C_VEL
LIN {X 0,Y 580.396,Z 572.328,A -85,B 0,C 180,E1 -1815.811,E2 -1815.811} C_VEL
LIN {X 0,Y 580.365,Z 564.477,A -85,B 0,C 180,E1 -1818.352,E2 -1818.352} C_VEL
LIN {X 0,Y 580.24,Z 554.638,A -85,B 0,C 180,E1 -1821.307,E2 -1821.307} C_VEL
LIN {X 0,Y 580.235,Z 552.212,A -85,B 0,C 180,E1 -1822.054,E2 -1822.054} C_VEL
LIN {X 0,Y 580.316,Z 552.202,A -85,B 0,C 180,E1 -1824.731,E2 -1824.731} C_VEL
LIN {X 0,Y 580.287,Z 552.204,A -85,B 0,C 180,E1 -1827.402,E2 -1827.402} C_VEL
LIN {X 0,Y 580.292,Z 552.204,A -85,B 0,C 180,E1 -1829.773,E2 -1829.773} C_VEL
LIN {X 0,Y 580.301,Z 552.205,A -85,B 0,C 180,E1 -1832.201,E2 -1832.201} C_VEL
LIN {X 0,Y 580.298,Z 552.203,A -85,B 0,C 180,E1 -1834.696,E2 -1834.696} C_VEL
LIN {X 0,Y 580.296,Z 552.204,A -85,B 0,C 180,E1 -1837.269,E2 -1837.269} C_VEL
LIN {X 0,Y 580.296,Z 552.203,A -85,B 0,C 180,E1 -1840.272,E2 -1840.272} C_VEL
LIN {X 0,Y 580.277,Z 552.207,A -85,B 0,C 180,E1 -1842.707,E2 -1842.707} C_VEL
LIN {X 0,Y 580.27,Z 552.208,A -85,B 0,C 180,E1 -1845.609,E2 -1845.609} C_VEL
LIN {X 0,Y 580.311,Z 552.201,A -85,B 0,C 180,E1 -1848.235,E2 -1848.235} C_VEL
LIN {X 0,Y 580.289,Z 552.206,A -85,B 0,C 180,E1 -1850.967,E2 -1850.967} C_VEL
LIN {X 0,Y 580.325,Z 552.238,A -85,B 0,C 180,E1 -1853.506,E2 -1853.506} C_VEL
LIN {X 0,Y 580.998,Z 556.972,A -85,B 0,C 180,E1 -1854.506,E2 -1854.506} C_VEL
LIN {X 0,Y 581.061,Z 571.781,A -85,B 0,C 180,E1 -1857.438,E2 -1857.438} C_VEL
LIN {X 0,Y 581.08,Z 586.675,A -85,B 0,C 180,E1 -1860.273,E2 -1860.273} C_VEL
LIN {X 0,Y 580.904,Z 600.425,A -85,B 0,C 180,E1 -1863.02,E2 -1863.02} C_VEL
LIN {X 0,Y 580.772,Z 614.175,A -85,B 0,C 180,E1 -1865.706,E2 -1865.706} C_VEL
LIN {X 0,Y 580.6,Z 630.162,A -85,B 0,C 180,E1 -1868.759,E2 -1868.759} C_VEL
LIN {X 0,Y 580.47,Z 645.603,A -85,B 0,C 180,E1 -1871.653,E2 -1871.653} C_VEL
LIN {X 0,Y 580.349,Z 661.317,A -85,B 0,C 180,E1 -1874.55,E2 -1874.55} C_VEL
LIN {X 0,Y 580.269,Z 677.031,A -85,B 0,C 180,E1 -1877.409,E2 -1877.409} C_VEL
LIN {X 0,Y 580.272,Z 678.139,A -85,B 0,C 180,E1 -1877.609,E2 -1877.609} C_VEL
LIN {X 0,Y 580.805,Z 683.985,A -85,B 0,C 180,E1 -1877.709,E2 -1877.709} C_VEL
LIN {X 0,Y 580.713,Z 697.244,A -85,B 0,C 180,E1 -1878.017,E2 -1878.017} C_VEL
LIN {X 0,Y 580.649,Z 710.511,A -85,B 0,C 180,E1 -1878.481,E2 -1878.481} C_VEL
LIN {X 0,Y 580.559,Z 721.645,A -85,B 0,C 180,E1 -1879.009,E2 -1879.009} C_VEL
LIN {X 0,Y 580.424,Z 733.212,A -85,B 0,C 180,E1 -1879.713,E2 -1879.713} C_VEL
LIN {X 0,Y 580.346,Z 743.606,A -85,B 0,C 180,E1 -1880.504,E2 -1880.504} C_VEL
LIN {X 0,Y 580.271,Z 752.119,A -85,B 0,C 180,E1 -1881.293,E2 -1881.293} C_VEL
LIN {X 0,Y 580.221,Z 759.966,A -85,B 0,C 180,E1 -1882.169,E2 -1882.169} C_VEL
LIN {X 0,Y 580.153,Z 767.654,A -85,B 0,C 180,E1 -1883.222,E2 -1883.222} C_VEL
LIN {X 0,Y 580.139,Z 774.684,A -85,B 0,C 180,E1 -1884.439,E2 -1884.439} C_VEL
LIN {X 0,Y 580.108,Z 779.374,A -85,B 0,C 180,E1 -1885.484,E2 -1885.484} C_VEL
LIN {X 0,Y 580.123,Z 782.959,A -85,B 0,C 180,E1 -1886.528,E2 -1886.528} C_VEL
LIN {X 0,Y 580.043,Z 784.81,A -85,B 0,C 180,E1 -1887.223,E2 -1887.223} C_VEL
LIN {X 0,Y 580.038,Z 786.201,A -85,B 0,C 180,E1 -1887.918,E2 -1887.918} C_VEL
LIN {X 0,Y 580.04,Z 787.785,A -85,B 0,C 180,E1 -1889.306,E2 -1889.306} C_VEL
LIN {X 0,Y 580.037,Z 788,A -85,B 0,C 180,E1 -1890.001,E2 -1890.001} C_VEL
LIN {X 0,Y 580.047,Z 787.185,A -85,B 0,C 180,E1 -1891.389,E2 -1891.389} C_VEL
LIN {X 0,Y 580.038,Z 786.2,A -85,B 0,C 180,E1 -1892.084,E2 -1892.084} C_VEL
LIN {X 0,Y 580.043,Z 784.808,A -85,B 0,C 180,E1 -1892.779,E2 -1892.779} C_VEL
LIN {X 0,Y 580.109,Z 781.894,A -85,B 0,C 180,E1 -1893.821,E2 -1893.821} C_VEL
LIN {X 0,Y 580.054,Z 777.947,A -85,B 0,C 180,E1 -1894.866,E2 -1894.866} C_VEL
LIN {X 0,Y 580.139,Z 771.874,A -85,B 0,C 180,E1 -1896.085,E2 -1896.085} C_VEL
LIN {X 0,Y 580.185,Z 765.232,A -85,B 0,C 180,E1 -1897.133,E2 -1897.133} C_VEL
LIN {X 0,Y 580.251,Z 756.985,A -85,B 0,C 180,E1 -1898.182,E2 -1898.182} C_VEL
LIN {X 0,Y 580.308,Z 748.531,A -85,B 0,C 180,E1 -1899.059,E2 -1899.059} C_VEL
LIN {X 0,Y 580.415,Z 738.087,A -85,B 0,C 180,E1 -1899.937,E2 -1899.937} C_VEL
LIN {X 0,Y 580.522,Z 727.749,A -85,B 0,C 180,E1 -1900.64,E2 -1900.64} C_VEL
LIN {X 0,Y 580.574,Z 716.581,A -85,B 0,C 180,E1 -1901.248,E2 -1901.248} C_VEL
LIN {X 0,Y 580.664,Z 704.751,A -85,B 0,C 180,E1 -1901.741,E2 -1901.741} C_VEL
LIN {X 0,Y 580.756,Z 691.327,A -85,B 0,C 180,E1 -1902.138,E2 -1902.138} C_VEL
LIN {X 0,Y 580.628,Z 680.694,A -85,B 0,C 180,E1 -1902.346,E2 -1902.346} C_VEL
LIN {X 0,Y 580.255,Z 678.031,A -85,B 0,C 180,E1 -1902.415,E2 -1902.415} C_VEL
LIN {X 0,Y 580.343,Z 663.358,A -85,B 0,C 180,E1 -1905.092,E2 -1905.092} C_VEL
LIN {X 0,Y 580.439,Z 647.707,A -85,B 0,C 180,E1 -1907.985,E2 -1907.985} C_VEL
LIN {X 0,Y 580.588,Z 632.198,A -85,B 0,C 180,E1 -1910.895,E2 -1910.895} C_VEL
LIN {X 0,Y 580.723,Z 616.404,A -85,B 0,C 180,E1 -1913.918,E2 -1913.918} C_VEL
LIN {X 0,Y 580.885,Z 602.71,A -85,B 0,C 180,E1 -1916.594,E2 -1916.594} C_VEL
LIN {X 0,Y 581.06,Z 588.47,A -85,B 0,C 180,E1 -1919.442,E2 -1919.442} C_VEL
LIN {X 0,Y 581.029,Z 575.538,A -85,B 0,C 180,E1 -1921.943,E2 -1921.943} C_VEL
LIN {X 0,Y 581.021,Z 562.802,A -85,B 0,C 180,E1 -1924.436,E2 -1924.436} C_VEL
LIN {X 0,Y 580.839,Z 554.907,A -85,B 0,C 180,E1 -1926.069,E2 -1926.069} C_VEL
LIN {X 0,Y 580.319,Z 552.201,A -85,B 0,C 180,E1 -1926.686,E2 -1926.686} C_VEL
LIN {X 0,Y 580.314,Z 552.2,A -85,B 0,C 180,E1 -1929.187,E2 -1929.187} C_VEL
LIN {X 0,Y 580.319,Z 552.2,A -85,B 0,C 180,E1 -1931.766,E2 -1931.766} C_VEL
LIN {X 0,Y 580.272,Z 552.207,A -85,B 0,C 180,E1 -1934.626,E2 -1934.626} C_VEL
LIN {X 0,Y 580.292,Z 552.203,A -85,B 0,C 180,E1 -1937.628,E2 -1937.628} C_VEL
LIN {X 0,Y 580.288,Z 552.204,A -85,B 0,C 180,E1 -1940.066,E2 -1940.066} C_VEL
LIN {X 0,Y 580.306,Z 552.2,A -85,B 0,C 180,E1 -1943.065,E2 -1943.065} C_VEL
LIN {X 0,Y 580.308,Z 552.2,A -85,B 0,C 180,E1 -1945.441,E2 -1945.441} C_VEL
LIN {X 0,Y 580.305,Z 552.201,A -85,B 0,C 180,E1 -1947.969,E2 -1947.969} C_VEL
LIN {X 0,Y 580.306,Z 552.203,A -85,B 0,C 180,E1 -1950.69,E2 -1950.69} C_VEL
LIN {X 0,Y 580.282,Z 552.205,A -85,B 0,C 180,E1 -1953.377,E2 -1953.377} C_VEL
LIN {X 0,Y 580.304,Z 552.203,A -85,B 0,C 180,E1 -1955.684,E2 -1955.684} C_VEL
LIN {X 0,Y 580.278,Z 552.206,A -85,B 0,C 180,E1 -1957.947,E2 -1957.947} C_VEL
LIN {X 0,Y 580.324,Z 552.199,A -85,B 0,C 180,E1 -1960.914,E2 -1960.914} C_VEL
LIN {X 0,Y 580.284,Z 552.205,A -85,B 0,C 180,E1 -1963.825,E2 -1963.825} C_VEL
LIN {X 0,Y 580.329,Z 552.201,A -85,B 0,C 180,E1 -1965.983,E2 -1965.983} C_VEL
LIN {X 0,Y 580.309,Z 552.2,A -85,B 0,C 180,E1 -1968.827,E2 -1968.827} C_VEL
LIN {X 0,Y 580.337,Z 552.198,A -85,B 0,C 180,E1 -1971.644,E2 -1971.644} C_VEL
LIN {X 0,Y 580.326,Z 552.199,A -85,B 0,C 180,E1 -1974.44,E2 -1974.44} C_VEL
LIN {X 0,Y 580.344,Z 552.196,A -85,B 0,C 180,E1 -1977.223,E2 -1977.223} C_VEL
LIN {X 0,Y 580.356,Z 552.198,A -85,B 0,C 180,E1 -1980,E2 -1980} C_VEL
LIN {X 0,Y 580.344,Z 552.196,A -85,B 0,C 180,E1 -1982.776,E2 -1982.776} C_VEL
LIN {X 0,Y 580.325,Z 552.199,A -85,B 0,C 180,E1 -1985.559,E2 -1985.559} C_VEL
LIN {X 0,Y 580.332,Z 552.199,A -85,B 0,C 180,E1 -1988.356,E2 -1988.356} C_VEL
LIN {X 0,Y 580.303,Z 552.201,A -85,B 0,C 180,E1 -1991.191,E2 -1991.191} C_VEL
LIN {X 0,Y 580.33,Z 552.201,A -85,B 0,C 180,E1 -1994.017,E2 -1994.017} C_VEL
LIN {X 0,Y 580.315,Z 552.2,A -85,B 0,C 180,E1 -1996.913,E2 -1996.913} C_VEL
LIN {X 0,Y 580.306,Z 552.203,A -85,B 0,C 180,E1 -1999.822,E2 -1999.822} C_VEL
LIN {X 0,Y 580.286,Z 552.204,A -85,B 0,C 180,E1 -2001.332,E2 -2001.332} C_VEL
LIN {X 0,Y 579.59,Z 552.291,A -85,B 0,C 180,E1 -2001.911,E2 -2001.911} C_VEL
LIN {X 0,Y 576.713,Z 552.648,A -85,B 0,C 180,E1 -2002.851,E2 -2002.851} C_VEL
LIN {X 0,Y 574.318,Z 552.948,A -85,B 0,C 180,E1 -2003.607,E2 -2003.607} C_VEL
LIN {X 0,Y 573.319,Z 553.072,A -85,B 0,C 180,E1 -2004.191,E2 -2004.191} C_VEL
LIN {X 0,Y 573.252,Z 553.079,A -85,B 0,C 180,E1 -2004.389,E2 -2004.389} C_VEL
LIN {X 0,Y 573.253,Z 553.081,A -85,B 0,C 180,E1 -2006.975,E2 -2006.975} C_VEL
LIN {X 0,Y 573.25,Z 553.08,A -85,B 0,C 180,E1 -2009.488,E2 -2009.488} C_VEL
LIN {X 0,Y 573.255,Z 553.082,A -85,B 0,C 180,E1 -2012.645,E2 -2012.645} C_VEL
LIN {X 0,Y 573.27,Z 553.079,A -85,B 0,C 180,E1 -2015.183,E2 -2015.183} C_VEL
LIN {X 0,Y 573.237,Z 553.081,A -85,B 0,C 180,E1 -2017.807,E2 -2017.807} C_VEL
LIN {X 0,Y 573.271,Z 553.078,A -85,B 0,C 180,E1 -2020.528,E2 -2020.528} C_VEL
LIN {X 0,Y 573.254,Z 553.079,A -85,B 0,C 180,E1 -2023.669,E2 -2023.669} C_VEL
LIN {X 0,Y 573.248,Z 553.083,A -85,B 0,C 180,E1 -2026.641,E2 -2026.641} C_VEL
LIN {X 0,Y 573.275,Z 553.076,A -85,B 0,C 180,E1 -2029.477,E2 -2029.477} C_VEL
LIN {X 0,Y 573.238,Z 553.081,A -85,B 0,C 180,E1 -2032.192,E2 -2032.192} C_VEL
LIN {X 0,Y 573.236,Z 553.081,A -85,B 0,C 180,E1 -2035.228,E2 -2035.228} C_VEL
LIN {X 0,Y 573.258,Z 553.078,A -85,B 0,C 180,E1 -2037.77,E2 -2037.77} C_VEL
LIN {X 0,Y 573.265,Z 553.08,A -85,B 0,C 180,E1 -2040.634,E2 -2040.634} C_VEL
LIN {X 0,Y 573.253,Z 553.083,A -85,B 0,C 180,E1 -2043.024,E2 -2043.024} C_VEL
LIN {X 0,Y 573.276,Z 553.079,A -85,B 0,C 180,E1 -2045.366,E2 -2045.366} C_VEL
LIN {X 0,Y 573.23,Z 553.082,A -85,B 0,C 180,E1 -2048.419,E2 -2048.419} C_VEL
LIN {X 0,Y 573.279,Z 553.076,A -85,B 0,C 180,E1 -2050.728,E2 -2050.728} C_VEL
LIN {X 0,Y 573.253,Z 553.082,A -85,B 0,C 180,E1 -2053.621,E2 -2053.621} C_VEL
LIN {X 0,Y 573.274,Z 553.079,A -85,B 0,C 180,E1 -2055.806,E2 -2055.806} C_VEL
LIN {X 0,Y 573.263,Z 553.078,A -85,B 0,C 180,E1 -2058.744,E2 -2058.744} C_VEL
LIN {X 0,Y 573.284,Z 553.077,A -85,B 0,C 180,E1 -2061.54,E2 -2061.54} C_VEL
LIN {X 0,Y 573.291,Z 553.076,A -85,B 0,C 180,E1 -2064.371,E2 -2064.371} C_VEL
LIN {X 0,Y 573.313,Z 553.073,A -85,B 0,C 180,E1 -2067.892,E2 -2067.892} C_VEL
LIN {X 0,Y 573.328,Z 553.071,A -85,B 0,C 180,E1 -2070.702,E2 -2070.702} C_VEL
LIN {X 0,Y 573.312,Z 553.074,A -85,B 0,C 180,E1 -2072.085,E2 -2072.085} C_VEL
LIN {X 0,Y 573.69,Z 557.944,A -85,B 0,C 180,E1 -2072.281,E2 -2072.281} C_VEL
LIN {X 0,Y 573.597,Z 569.482,A -85,B 0,C 180,E1 -2072.809,E2 -2072.809} C_VEL
LIN {X 0,Y 573.452,Z 580.071,A -85,B 0,C 180,E1 -2073.425,E2 -2073.425} C_VEL
LIN {X 0,Y 573.361,Z 589.873,A -85,B 0,C 180,E1 -2074.129,E2 -2074.129} C_VEL
LIN {X 0,Y 573.257,Z 598.971,A -85,B 0,C 180,E1 -2074.922,E2 -2074.922} C_VEL
LIN {X 0,Y 573.144,Z 607.351,A -85,B 0,C 180,E1 -2075.805,E2 -2075.805} C_VEL
LIN {X 0,Y 573.111,Z 615.749,A -85,B 0,C 180,E1 -2076.895,E2 -2076.895} C_VEL
LIN {X 0,Y 573.043,Z 623.061,A -85,B 0,C 180,E1 -2078.107,E2 -2078.107} C_VEL
LIN {X 0,Y 572.989,Z 628.127,A -85,B 0,C 180,E1 -2079.174,E2 -2079.174} C_VEL
LIN {X 0,Y 572.99,Z 632.057,A -85,B 0,C 180,E1 -2080.244,E2 -2080.244} C_VEL
LIN {X 0,Y 572.971,Z 634.949,A -85,B 0,C 180,E1 -2081.317,E2 -2081.317} C_VEL
LIN {X 0,Y 572.944,Z 636.361,A -85,B 0,C 180,E1 -2082.035,E2 -2082.035} C_VEL
LIN {X 0,Y 572.944,Z 637.31,A -85,B 0,C 180,E1 -2082.755,E2 -2082.755} C_VEL
LIN {X 0,Y 572.972,Z 637.972,A -85,B 0,C 180,E1 -2084.2,E2 -2084.2} C_VEL
LIN {X 0,Y 572.904,Z 637.666,A -85,B 0,C 180,E1 -2084.928,E2 -2084.928} C_VEL
LIN {X 0,Y 572.948,Z 635.773,A -85,B 0,C 180,E1 -2086.386,E2 -2086.386} C_VEL
LIN {X 0,Y 572.97,Z 633.16,A -85,B 0,C 180,E1 -2087.488,E2 -2087.488} C_VEL
LIN {X 0,Y 573.005,Z 629.435,A -85,B 0,C 180,E1 -2088.595,E2 -2088.595} C_VEL
LIN {X 0,Y 573.051,Z 624.464,A -85,B 0,C 180,E1 -2089.709,E2 -2089.709} C_VEL
